(* IEC 61131-3 sources: Supremica/tests/ilprograms, 8 files *)

(* ---- arithmetictest.il ---- *)
(* Must test EQ before this.
 *)
PROGRAM ArithmeticTest
   VAR
	BB1, BB2, BB3 : BOOL;
	DD1, DD2, DD3 : DINT;
	RR1, RR2, RR3 : REAL;
	WW1, WW2, WW3 : WSTRING;
   END_VAR
   VAR
	Assert   : Asserter;
	(*Printing*)
	WPrintln : PrintlnWSTRING;
	DPrintln : PrintlnDINT;
	BPrintln : PrintlnBOOL;
	RPrintln : PrintlnREAL;
	WPrint   : PrintWSTRING;
	DPrint   : PrintDINT;
	BPrint   : PrintBOOL;
	RPrint   : PrintREAL;
   END_VAR

CAL WPrintln("Testing ADD")
	CAL Assert(TRUE,"här skall INGET fel ges")
	CAL Assert(FALSE,"här skall ett fel ges")
CAL WPrintln("Testing SUB")

CAL WPrintln("Testing MUL")

CAL WPrintln("Testing DIV")

CAL WPrintln("Testing MOD")

END_PROGRAM

FUNCTION_BLOCK Asserter
	VAR_IN_OUT
		result : BOOL;
		msg    : WSTRING;
	END_VAR
	VAR
		WPrintln : PrintlnWSTRING;
		WPrint   : PrintWSTRING;
	END_VAR
	LD result
	JMPC noerror
		CAL WPrint(output := "fdsf")
		(*CAL WPrint("Error: assertion not true! : ")*)
		(*CAL WPrintln(msg)*)
noerror:
END_FUNCTION_BLOCK

(*JAVA_BLOCKS for printing (no newline)*)
(*=====================================*)

JAVA_BLOCK JPrintWSTRING
	VAR_IN_OUT
		output: WSTRING;
	END_VAR
END_JAVA_BLOCK
FUNCTION_BLOCK PrintWSTRING
	VAR_IN_OUT
		output: WSTRING;
	END_VAR
	VAR
		jblock: JPrintWSTRING;
	END_VAR
	LD output
	ST jblock.output
	CAL jblock
END_FUNCTION_BLOCK

JAVA_BLOCK JPrintDINT
	VAR_IN_OUT
		output: DINT;
	END_VAR
END_JAVA_BLOCK
FUNCTION_BLOCK PrintDINT
	VAR_IN_OUT
		output: DINT;
	END_VAR
	VAR
		jblock: JPrintDINT;
	END_VAR
	LD output
	ST jblock.output
	CAL jblock
END_FUNCTION_BLOCK
JAVA_BLOCK JPrintREAL
	VAR_IN_OUT
		output:REAL;
	END_VAR
END_JAVA_BLOCK
FUNCTION_BLOCK PrintREAL
	VAR_IN_OUT
		output:REAL;
	END_VAR
	VAR
		jblock:JPrintREAL;
	END_VAR
	LD output
	ST jblock.output
	CAL jblock
END_FUNCTION_BLOCK

JAVA_BLOCK JPrintBOOL
	VAR_IN_OUT
		output: BOOL;
	END_VAR
END_JAVA_BLOCK
FUNCTION_BLOCK PrintBOOL
	VAR_IN_OUT
		output: BOOL;
	END_VAR
	VAR
		jblock: JPrintBOOL;
	END_VAR
	LD output
	ST jblock.output
	CAL jblock
END_FUNCTION_BLOCK

(*JAVA_BLOCKS for printing (newline)*)
(*=====================================*)

JAVA_BLOCK JPrintlnWSTRING
	VAR_IN_OUT
		output: WSTRING;
	END_VAR
END_JAVA_BLOCK
FUNCTION_BLOCK PrintlnWSTRING
	VAR_IN_OUT
		output: WSTRING;
	END_VAR
	VAR
		jblock: JPrintlnWSTRING;
	END_VAR
	LD output
	ST jblock.output
	CAL jblock
END_FUNCTION_BLOCK

JAVA_BLOCK JPrintlnDINT
	VAR_IN_OUT
		output: DINT;
	END_VAR
END_JAVA_BLOCK
FUNCTION_BLOCK PrintlnDINT
	VAR_IN_OUT
		output: DINT;
	END_VAR
	VAR
		jblock: JPrintlnDINT;
	END_VAR
	LD output
	ST jblock.output
	CAL jblock
END_FUNCTION_BLOCK

JAVA_BLOCK JPrintlnREAL
	VAR_IN_OUT
		output:REAL;
	END_VAR
END_JAVA_BLOCK
FUNCTION_BLOCK PrintlnREAL
	VAR_IN_OUT
		output:REAL;
	END_VAR
	VAR
		jblock:JPrintlnREAL;
	END_VAR
	LD output
	ST jblock.output
	CAL jblock
END_FUNCTION_BLOCK

JAVA_BLOCK JPrintlnBOOL
	VAR_IN_OUT
		output: BOOL;
	END_VAR
END_JAVA_BLOCK
FUNCTION_BLOCK PrintlnBOOL
	VAR_IN_OUT
		output: BOOL;
	END_VAR
	VAR
		jblock: JPrintlnBOOL;
	END_VAR
	LD output
	ST jblock.output
	CAL jblock
END_FUNCTION_BLOCK

(* ---- caltest.il ---- *)
(*JAVA_BLOCKS for printing (no newline)*)
(*=====================================*)

JAVA_BLOCK JPrintWSTRING
	VAR_IN_OUT
		output: WSTRING;
	END_VAR
END_JAVA_BLOCK
FUNCTION_BLOCK PrintWSTRING
	VAR_IN_OUT
		output: WSTRING;
	END_VAR
	VAR
		jblock: JPrintWSTRING;
	END_VAR
	LD output
	ST jblock.output
	CAL jblock
END_FUNCTION_BLOCK

JAVA_BLOCK JPrintDINT
	VAR_IN_OUT
		output: DINT;
	END_VAR
END_JAVA_BLOCK
FUNCTION_BLOCK PrintDINT
	VAR_IN_OUT
		output: DINT;
	END_VAR
	VAR
		jblock: JPrintDINT;
	END_VAR
	LD output
	ST jblock.output
	CAL jblock
END_FUNCTION_BLOCK

JAVA_BLOCK JPrintREAL
	VAR_IN_OUT
		output:REAL;
	END_VAR
END_JAVA_BLOCK
FUNCTION_BLOCK PrintREAL
	VAR_IN_OUT
		output:REAL;
	END_VAR
	VAR
		jblock:JPrintREAL;
	END_VAR
	LD output
	ST jblock.output
	CAL jblock
END_FUNCTION_BLOCK

JAVA_BLOCK JPrintBOOL
	VAR_IN_OUT
		output: BOOL;
	END_VAR
END_JAVA_BLOCK
FUNCTION_BLOCK PrintBOOL
	VAR_IN_OUT
		output: BOOL;
	END_VAR
	VAR
		jblock: JPrintBOOL;
	END_VAR
	LD output
	ST jblock.output
	CAL jblock
END_FUNCTION_BLOCK

(*JAVA_BLOCKS for printing (newline)*)
(*=====================================*)

JAVA_BLOCK JPrintlnWSTRING
	VAR_IN_OUT
		output: WSTRING;
	END_VAR
END_JAVA_BLOCK
FUNCTION_BLOCK PrintlnWSTRING
	VAR_IN_OUT
		output: WSTRING;
	END_VAR
	VAR
		jblock: JPrintlnWSTRING;
	END_VAR
	LD output
	ST jblock.output
	CAL jblock
END_FUNCTION_BLOCK

JAVA_BLOCK JPrintlnDINT
	VAR_IN_OUT
		output: DINT;
	END_VAR
END_JAVA_BLOCK
FUNCTION_BLOCK PrintlnDINT
	VAR_IN_OUT
		output: DINT;
	END_VAR
	VAR
		jblock: JPrintlnDINT;
	END_VAR
	LD output
	ST jblock.output
	CAL jblock
END_FUNCTION_BLOCK

JAVA_BLOCK JPrintlnREAL
	VAR_IN_OUT
		output:REAL;
	END_VAR
END_JAVA_BLOCK
FUNCTION_BLOCK PrintlnREAL
	VAR_IN_OUT
		output:REAL;
	END_VAR
	VAR
		jblock:JPrintlnREAL;
	END_VAR
	LD output
	ST jblock.output
	CAL jblock
END_FUNCTION_BLOCK

JAVA_BLOCK JPrintlnBOOL
	VAR_IN_OUT
		output: BOOL;
	END_VAR
END_JAVA_BLOCK
FUNCTION_BLOCK PrintlnBOOL
	VAR_IN_OUT
		output: BOOL;
	END_VAR
	VAR
		jblock: JPrintlnBOOL;
	END_VAR
	LD output
	ST jblock.output
	CAL jblock
END_FUNCTION_BLOCK

FUNCTION_BLOCK PrintlnWSTRING_DINT
	VAR_IN_OUT
		string: WSTRING;
		dint  : DINT;
	END_VAR
	VAR
		jblockWS: JPrintWSTRING;
		jblockD : JPrintlnDINT;
	END_VAR

	LD string
	ST jblockWS.output
	CAL jblockWS

	LD dint
	ST jblockD.output
	CAL jblockD
END_FUNCTION_BLOCK

FUNCTION_BLOCK DOUBLER
	VAR_IN_OUT
		A : DINT;
	END_VAR

	LD A
	ADD A

	ST A

END_FUNCTION_BLOCK

FUNCTION_BLOCK ADDER
	VAR_IN_OUT
		in_1 : DINT;
	    in_2 : DINT;
		out  : DINT;
	END_VAR

	LD in_1
	ADD in_2

	ST out

END_FUNCTION_BLOCK

FUNCTION_BLOCK ANDER
	VAR_IN_OUT
		in_1 : BOOL;
	    in_2 : BOOL;
		out  : BOOL;

	END_VAR

	LD in_1
	AND in_2
	ST out

END_FUNCTION_BLOCK

PROGRAM CALTEST
	VAR
		print_WS   : PrintWSTRING;
		print_DINT : PrintDINT;
		print_REAL : PrintREAL;
		print_BOOL : PrintBOOL;

		println_WS   : PrintlnWSTRING;
		println_DINT : PrintlnDINT;
		println_REAL : PrintlnREAL;
		println_BOOL : PrintlnBOOL;

		printlnWS_D  : PrintlnWSTRING_DINT;

      	doubler      : DOUBLER;
		adder        : ADDER;
		ander        : ANDER;

		N1           : DINT;
		N2           : DINT;
      	Result_DINT  : DINT;
		Result_BOOL  : BOOL;
	END_VAR
	VAR
		b AT %QX1 : BOOL;
	END_VAR

	LD FALSE
	ST %QX1

	LD %QX1
	ST Result_BOOL

	CAL println_BOOL(Result_BOOL)

	CAL println_BOOL(%QX1)

	LD DINT#10
	ST N1

	CAL printlnWS_D("Doubler input: ", N1)
    CAL doubler(N1)
	CAL printlnWS_D("Doubler output: ", doubler.A)

	CAL printlnWS_D("Doubler input: ", N1)
    CAL doubler(A:=N1)
	CAL printlnWS_D("Doubler output: ", doubler.A)

	CAL printlnWS_D("Doubler input: ", DINT#33)
    CAL doubler(DINT#33)
	CAL printlnWS_D("Doubler output: ", doubler.A)

	CAL printlnWS_D("Doubler input: ", DINT#33)
    CAL doubler(A:=DINT#33)
	CAL printlnWS_D("Doubler output: ", doubler.A)

	CAL adder(in_1:=DINT#100, in_2:=DINT#200, out=>Result_DINT)
	CAL println_DINT(Result_DINT)

	CAL ander(in_1:=FALSE, in_2:=TRUE, out=>%QX1)
	CAL println_BOOL(%QX1)

END_PROGRAM

(* ---- cmp_tests.il ---- *)
(*
Test av EQ, GT, GE, LT, LE, NE
*)

JAVA_BLOCK JPrintWSTRING
	VAR_IN_OUT
		output: WSTRING;
	END_VAR
END_JAVA_BLOCK
FUNCTION_BLOCK PrintWSTRING
	VAR_IN_OUT
		output: WSTRING;
	END_VAR
	VAR
		jblock: JPrintWSTRING;
	END_VAR
	LD output
	ST jblock.output
	CAL jblock
END_FUNCTION_BLOCK

JAVA_BLOCK JPrintDINT
	VAR_IN_OUT
		output: DINT;
	END_VAR
END_JAVA_BLOCK
FUNCTION_BLOCK PrintDINT
	VAR_IN_OUT
		output: DINT;
	END_VAR
	VAR
		jblock: JPrintDINT;
	END_VAR
	LD output
	ST jblock.output
	CAL jblock
END_FUNCTION_BLOCK
JAVA_BLOCK JPrintREAL
	VAR_IN_OUT
		output:REAL;
	END_VAR
END_JAVA_BLOCK
FUNCTION_BLOCK PrintREAL
	VAR_IN_OUT
		output:REAL;
	END_VAR
	VAR
		jblock:JPrintREAL;
	END_VAR
	LD output
	ST jblock.output
	CAL jblock
END_FUNCTION_BLOCK

JAVA_BLOCK JPrintBOOL
	VAR_IN_OUT
		output: BOOL;
	END_VAR
END_JAVA_BLOCK
FUNCTION_BLOCK PrintBOOL
	VAR_IN_OUT
		output: BOOL;
	END_VAR
	VAR
		jblock: JPrintBOOL;
	END_VAR
	LD output
	ST jblock.output
	CAL jblock
END_FUNCTION_BLOCK

JAVA_BLOCK JPrintlnWSTRING
	VAR_IN_OUT
		output: WSTRING;
	END_VAR
END_JAVA_BLOCK
FUNCTION_BLOCK PrintlnWSTRING
	VAR_IN_OUT
		output: WSTRING;
	END_VAR
	VAR
		jblock: JPrintlnWSTRING;
	END_VAR
	LD output
	ST jblock.output
	CAL jblock
END_FUNCTION_BLOCK

JAVA_BLOCK JPrintlnBOOL
	VAR_IN_OUT
		output: BOOL;
	END_VAR
END_JAVA_BLOCK
FUNCTION_BLOCK PrintlnBOOL
	VAR_IN_OUT
		output: BOOL;
	END_VAR
	VAR
		jblock: JPrintlnBOOL;
	END_VAR
	LD output
	ST jblock.output
	CAL jblock
END_FUNCTION_BLOCK

JAVA_BLOCK JPrintlnDINT
	VAR_IN_OUT
		output: DINT;
	END_VAR
END_JAVA_BLOCK
FUNCTION_BLOCK PrintlnDINT
	VAR_IN_OUT
		output: DINT;
	END_VAR
	VAR
		jblock: JPrintlnDINT;
	END_VAR
	LD output
	ST jblock.output
	CAL jblock
END_FUNCTION_BLOCK

JAVA_BLOCK JPrintlnREAL
	VAR_IN_OUT
		output:REAL;
	END_VAR
END_JAVA_BLOCK
FUNCTION_BLOCK PrintlnREAL
	VAR_IN_OUT
		output:REAL;
	END_VAR
	VAR
		jblock:JPrintlnREAL;
	END_VAR
	LD output
	ST jblock.output
	CAL jblock
END_FUNCTION_BLOCK

PROGRAM CMPtests
   VAR
	BB1, BB2, BB3 : BOOL;
	DD1, DD2, DD3 : DINT;
	RR1, RR2, RR3 : REAL;
	WW1, WW2, WW3 : WSTRING;
	PRINT_S : JPrintWSTRING;
	PRINT_B : JPrintBOOL;
	PRINT_I : JPrintDINT;
	PRINT_R : JPrintREAL;
	PRINTLN_S : JPrintlnWSTRING;
	PRINTLN_B : JPrintlnBOOL;
	PRINTLN_I : JPrintlnDINT;
	PRINTLN_R : JPrintlnREAL;
   END_VAR

	(*BOOL- jämför stack med variabel*)
	CAL PRINTLN_S(output:="EQ - BOOL")
(*T-T*)
	LD TRUE
	ST BB1
	LD TRUE
	EQ BB1
	ST BB2
	CAL PRINT_S(output:="?? true == ")
	CAL PRINTLN_B(output:=BB2)
(*T-F*)
	LD FALSE
	ST BB1
	LD TRUE
	EQ BB1
	ST BB2
	CAL PRINT_S(output:="?? false == ")
	CAL PRINTLN_B(output:=BB2)
(*F-T*)
	LD TRUE
	ST BB1
	LD FALSE
	EQ BB1
	ST BB2
	CAL PRINT_S(output:="?? false == ")
	CAL PRINTLN_B(output:=BB2)
(*F-F*)
	LD FALSE
	ST BB1
	LD FALSE
	EQ BB1
	ST BB2
	CAL PRINT_S(output:="?? true == ")
	CAL PRINTLN_B(output:=BB2)

	(*BOOL- jämför stack med konstant*)
(*T-T*)
	LD TRUE
	EQ TRUE
	ST BB2
	CAL PRINT_S(output:="?? true == ")
	CAL PRINTLN_B(output:=BB2)
(*T-F*)
	LD FALSE
	EQ TRUE
	ST BB2
	CAL PRINT_S(output:="?? false == ")
	CAL PRINTLN_B(output:=BB2)
(*F-T*)
	LD TRUE
	EQ FALSE
	ST BB2
	CAL PRINT_S(output:="?? false == ")
	CAL PRINTLN_B(output:=BB2)
(*F-F*)
	LD FALSE
	ST BB1
	LD FALSE
	EQ BB1
	ST BB2
	CAL PRINT_S(output:="?? true == ")
	CAL PRINTLN_B(output:=BB2)

	(*DINT - jämför stack med variabel*)
	CAL PRINTLN_S(output:="EQ - DINT")
(*1-1*)
	LD DINT#1
	ST DD1
	LD DINT#1
	EQ DD1
	ST BB2
	CAL PRINT_S(output:="?? true == ")
	CAL PRINTLN_B(output:=BB2)
(*2147483647 - 2147483647*)
	LD DINT#2147483647
	ST DD1
	LD DINT#2147483647
	EQ DD1
	ST BB2
	CAL PRINT_S(output:="?? true == ")
	CAL PRINTLN_B(output:=BB2)
(*-2147483647 - -2147483647*)
	LD DINT#-2147483647
	ST DD1
	LD DINT#-2147483647
	EQ DD1
	ST BB2
	CAL PRINT_S(output:="?? true == ")
	CAL PRINTLN_B(output:=BB2)
(*0 - 2147483647*)
	LD DINT#2147483647
	ST DD1
	LD DINT#0
	EQ DD1
	ST BB2
	CAL PRINT_S(output:="?? false == ")
	CAL PRINTLN_B(output:=BB2)
(*0 - -2147483647*)
	LD DINT#-2147483647
	ST DD1
	LD DINT#0
	EQ DD1
	ST BB2
	CAL PRINT_S(output:="?? false == ")
	CAL PRINTLN_B(output:=BB2)
(*-2147483647 - 0*)
	LD DINT#0
	ST DD1
	LD DINT#-2147483647
	EQ DD1
	ST BB2
	CAL PRINT_S(output:="?? false == ")
	CAL PRINTLN_B(output:=BB2)
(*2147483647 - 0*)
	LD DINT#0
	ST DD1
	LD DINT#2147483647
	EQ DD1
	ST BB2
	CAL PRINT_S(output:="?? false == ")
	CAL PRINTLN_B(output:=BB2)

	(*DINT- jämför stack med konstant*)
(*1-1*)
	LD DINT#1
	EQ DINT#1
	ST BB2
	CAL PRINT_S(output:="?? true == ")
	CAL PRINTLN_B(output:=BB2)
(*2147483647 - 2147483647*)
	LD DINT#2147483647
	EQ DINT#2147483647
	ST BB2
	CAL PRINT_S(output:="?? true == ")
	CAL PRINTLN_B(output:=BB2)
(*-2147483647 - -2147483647*)
	LD DINT#-2147483647
	EQ DINT#-2147483647
	ST BB2
	CAL PRINT_S(output:="?? true == ")
	CAL PRINTLN_B(output:=BB2)
(*0 - -2147483647*)
	LD DINT#2147483647
	EQ DINT#0
	ST BB2
	CAL PRINT_S(output:="?? false == ")
	CAL PRINTLN_B(output:=BB2)
(*0 - -2147483647*)
	LD DINT#-2147483647
	EQ DINT#0
	ST BB2
	CAL PRINT_S(output:="?? false == ")
	CAL PRINTLN_B(output:=BB2)
(*-2147483647 - 0*)
	LD DINT#0
	EQ DINT#-2147483647
	ST BB2
	CAL PRINT_S(output:="?? false == ")
	CAL PRINTLN_B(output:=BB2)
(*2147483647 - 0*)
	LD DINT#0
	EQ DINT#2147483647
	ST BB2
	CAL PRINT_S(output:="?? false == ")
	CAL PRINTLN_B(output:=BB2)

	(*EQ - REAL - jämför stack med variabel*)
	CAL PRINTLN_S(output:="EQ - REAL")
(*1.0 - 1.0*)
	LD REAL#1.0
	ST RR1
	LD REAL#1.0
	EQ RR1
	ST BB2
	CAL PRINT_S(output:="?? true == ")
	CAL PRINTLN_B(output:=BB2)
(*3.4028235E38 - 3.4028235E38*)
	LD REAL#3.4028235E38
	ST RR1
	LD REAL#3.4028235E38
	EQ RR1
	ST BB2
	CAL PRINT_S(output:="?? true == ")
	CAL PRINTLN_B(output:=BB2)
(*1.4E-45 - 1.4E-45*)
	LD REAL#1.4E-45
	ST RR1
	LD REAL#1.4E-45
	EQ RR1
	ST BB2
	CAL PRINT_S(output:="?? true == ")
	CAL PRINTLN_B(output:=BB2)
(*0 - 3.4028235E38*)
	LD REAL#3.4028235E38
	ST RR1
	LD REAL#0.0
	EQ RR1
	ST BB2
	CAL PRINT_S(output:="?? false == ")
	CAL PRINTLN_B(output:=BB2)
(*0 - 1.4E-45*)
	LD REAL#1.4E-45
	ST RR1
	LD REAL#0.0
	EQ RR1
	ST BB2
	CAL PRINT_S(output:="?? false == ")
	CAL PRINTLN_B(output:=BB2)
(*1.4E-45 - 0*)
	LD REAL#0.0
	ST RR1
	LD REAL#1.4E-45
	EQ RR1
	ST BB2
	CAL PRINT_S(output:="?? false == ")
	CAL PRINTLN_B(output:=BB2)
(*3.4028235E38 - 0*)
	LD REAL#0.0
	ST RR1
	LD REAL#3.4028235E38
	EQ RR1
	ST BB2
	CAL PRINT_S(output:="?? false == ")
	CAL PRINTLN_B(output:=BB2)

	(*EQ - REAL- jämför stack med konstant*)
(*1-1*)
	LD REAL#1.0
	EQ REAL#1.0
	ST BB2
	CAL PRINT_S(output:="?? true == ")
	CAL PRINTLN_B(output:=BB2)
(*3.4028235E38 - 3.4028235E38*)
	LD REAL#3.4028235E38
	EQ REAL#3.4028235E38
	ST BB2
	CAL PRINT_S(output:="?? true == ")
	CAL PRINTLN_B(output:=BB2)
(*1.4E-45 - 1.4E-45*)
	LD REAL#1.4E-45
	EQ REAL#1.4E-45
	ST BB2
	CAL PRINT_S(output:="?? true == ")
	CAL PRINTLN_B(output:=BB2)
(*0 - 3.4028235E38*)
	LD REAL#3.4028235E38
	EQ REAL#0.0
	ST BB2
	CAL PRINT_S(output:="?? false == ")
	CAL PRINTLN_B(output:=BB2)
(*0 - 1.4E-45*)
	LD REAL#1.4E-45
	EQ REAL#0.0
	ST BB2
	CAL PRINT_S(output:="?? false == ")
	CAL PRINTLN_B(output:=BB2)
(*1.4E-45 - 0*)
	LD REAL#0.0
	EQ REAL#1.4E-45
	ST BB2
	CAL PRINT_S(output:="?? false == ")
	CAL PRINTLN_B(output:=BB2)
(*3.4028235E38 - 0*)
	LD REAL#0.0
	EQ REAL#3.4028235E38
	ST BB2
	CAL PRINT_S(output:="?? false == ")
	CAL PRINTLN_B(output:=BB2)

(******************************************************************)

	(*GT - DINT - jämför stack med variabel*)
	CAL PRINTLN_S(output:="GT - DINT")
(*1-1*)
	LD DINT#1
	ST DD1
	LD DINT#1
	GT DD1
	ST BB2
	CAL PRINT_S(output:="?? false == ")
	CAL PRINTLN_B(output:=BB2)
(*2147483647 - 2147483647*)
	LD DINT#2147483647
	ST DD1
	LD DINT#2147483647
	GT DD1
	ST BB2
	CAL PRINT_S(output:="?? false == ")
	CAL PRINTLN_B(output:=BB2)
(*-2147483647 - -2147483647*)
	LD DINT#-2147483647
	ST DD1
	LD DINT#-2147483647
	GT DD1
	ST BB2
	CAL PRINT_S(output:="?? false == ")
	CAL PRINTLN_B(output:=BB2)
(*0 - 2147483647*)
	LD DINT#2147483647
	ST DD1
	LD DINT#0
	GT DD1
	ST BB2
	CAL PRINT_S(output:="?? false == ")
	CAL PRINTLN_B(output:=BB2)
(*0 - -2147483647*)
	LD DINT#-2147483647
	ST DD1
	LD DINT#0
	GT DD1
	ST BB2
	CAL PRINT_S(output:="?? true == ")
	CAL PRINTLN_B(output:=BB2)
(*-2147483647 - 0*)
	LD DINT#0
	ST DD1
	LD DINT#-2147483647
	GT DD1
	ST BB2
	CAL PRINT_S(output:="?? false == ")
	CAL PRINTLN_B(output:=BB2)
(*2147483647 - 0*)
	LD DINT#0
	ST DD1
	LD DINT#2147483647
	GT DD1
	ST BB2
	CAL PRINT_S(output:="?? true == ")
	CAL PRINTLN_B(output:=BB2)

	(*GT - DINT - jämför stack med konstant*)
(*1-1*)
	LD DINT#1
	GT DINT#1
	ST BB2
	CAL PRINT_S(output:="?? false == ")
	CAL PRINTLN_B(output:=BB2)
(*2147483647 - 2147483647*)
	LD DINT#2147483647
	GT DINT#2147483647
	ST BB2
	CAL PRINT_S(output:="?? false == ")
	CAL PRINTLN_B(output:=BB2)
(*-2147483647 - -2147483647*)
	LD DINT#-2147483647
	GT DINT#-2147483647
	ST BB2
	CAL PRINT_S(output:="?? false == ")
	CAL PRINTLN_B(output:=BB2)
(*2147483647 - 0*)
	LD DINT#2147483647
	GT DINT#0
	ST BB2
	CAL PRINT_S(output:="?? true == ")
	CAL PRINTLN_B(output:=BB2)
(*-2147483647 - 0*)
	LD DINT#-2147483647
	GT DINT#0
	ST BB2
	CAL PRINT_S(output:="?? false == ")
	CAL PRINTLN_B(output:=BB2)
(*0 - -2147483647*)
	LD DINT#0
	GT DINT#-2147483647
	ST BB2
	CAL PRINT_S(output:="?? true == ")
	CAL PRINTLN_B(output:=BB2)
(*0 - 2147483647*)
	LD DINT#0
	GT DINT#2147483647
	ST BB2
	CAL PRINT_S(output:="?? false == ")
	CAL PRINTLN_B(output:=BB2)

	(*GT - REAL - jämför stack med variabel*)
	CAL PRINTLN_S(output:="GT - REAL")
(*1.0 - 1.0*)
	LD REAL#1.0
	ST RR1
	LD REAL#1.0
	GT RR1
	ST BB2
	CAL PRINT_S(output:="?? false == ")
	CAL PRINTLN_B(output:=BB2)
(*3.4028235E38 - 3.4028235E38*)
	LD REAL#3.4028235E38
	ST RR1
	LD REAL#3.4028235E38
	GT RR1
	ST BB2
	CAL PRINT_S(output:="?? false == ")
	CAL PRINTLN_B(output:=BB2)
(*1.4E-45 - 1.4E-45*)
	LD REAL#1.4E-45
	ST RR1
	LD REAL#1.4E-45
	GT RR1
	ST BB2
	CAL PRINT_S(output:="?? false == ")
	CAL PRINTLN_B(output:=BB2)
(*0 - 3.4028235E38*)
	LD REAL#3.4028235E38
	ST RR1
	LD REAL#0.0
	GT RR1
	ST BB2
	CAL PRINT_S(output:="?? false == ")
	CAL PRINTLN_B(output:=BB2)
(*0 - 1.4E-45*)
	LD REAL#1.4E-45
	ST RR1
	LD REAL#0.0
	GT RR1
	ST BB2
	CAL PRINT_S(output:="?? false == ")
	CAL PRINTLN_B(output:=BB2)
(*1.4E-45 - 0*)
	LD REAL#0.0
	ST RR1
	LD REAL#1.4E-45
	GT RR1
	ST BB2
	CAL PRINT_S(output:="?? true == ")
	CAL PRINTLN_B(output:=BB2)
(*3.4028235E38 - 0*)
	LD REAL#0.0
	ST RR1
	LD REAL#3.4028235E38
	GT RR1
	ST BB2
	CAL PRINT_S(output:="?? true == ")
	CAL PRINTLN_B(output:=BB2)

	(*GT - REAL - jämför stack med konstant*)
(*1-1*)
	LD REAL#1.0
	GT REAL#1.0
	ST BB2
	CAL PRINT_S(output:="?? false == ")
	CAL PRINTLN_B(output:=BB2)
(*3.4028235E38 - 3.4028235E38*)
	LD REAL#3.4028235E38
	GT REAL#3.4028235E38
	ST BB2
	CAL PRINT_S(output:="?? false == ")
	CAL PRINTLN_B(output:=BB2)
(*1.4E-45 - 1.4E-45*)
	LD REAL#1.4E-45
	GT REAL#1.4E-45
	ST BB2
	CAL PRINT_S(output:="?? false == ")
	CAL PRINTLN_B(output:=BB2)
(*3.4028235E38 - 0*)
	LD REAL#3.4028235E38
	GT REAL#0.0
	ST BB2
	CAL PRINT_S(output:="?? true == ")
	CAL PRINTLN_B(output:=BB2)
(*1.4E-45 - 0*)
	LD REAL#1.4E-45
	GT REAL#0.0
	ST BB2
	CAL PRINT_S(output:="?? true == ")
	CAL PRINTLN_B(output:=BB2)
(*0 - 1.4E-45*)
	LD REAL#0.0
	GT REAL#1.4E-45
	ST BB2
	CAL PRINT_S(output:="?? false == ")
	CAL PRINTLN_B(output:=BB2)
(*0 - 3.4028235E38*)
	LD REAL#0.0
	GT REAL#3.4028235E38
	ST BB2
	CAL PRINT_S(output:="?? false == ")
	CAL PRINTLN_B(output:=BB2)

(*****************************************************************)

	(*GE - DINT - jämför stack med variabel*)
	CAL PRINTLN_S(output:="GE - DINT")
(*1-1*)
	LD DINT#1
	ST DD1
	LD DINT#1
	GE DD1
	ST BB2
	CAL PRINT_S(output:="?? true == ")
	CAL PRINTLN_B(output:=BB2)
(*2147483647 - 2147483647*)
	LD DINT#2147483647
	ST DD1
	LD DINT#2147483647
	GE DD1
	ST BB2
	CAL PRINT_S(output:="?? true == ")
	CAL PRINTLN_B(output:=BB2)
(*-2147483647 - -2147483647*)
	LD DINT#-2147483647
	ST DD1
	LD DINT#-2147483647
	GE DD1
	ST BB2
	CAL PRINT_S(output:="?? true == ")
	CAL PRINTLN_B(output:=BB2)
(*0 - 2147483647*)
	LD DINT#2147483647
	ST DD1
	LD DINT#0
	GE DD1
	ST BB2
	CAL PRINT_S(output:="?? false == ")
	CAL PRINTLN_B(output:=BB2)
(*0 - -2147483647*)
	LD DINT#-2147483647
	ST DD1
	LD DINT#0
	GE DD1
	ST BB2
	CAL PRINT_S(output:="?? true == ")
	CAL PRINTLN_B(output:=BB2)
(*-2147483647 - 0*)
	LD DINT#0
	ST DD1
	LD DINT#-2147483647
	GE DD1
	ST BB2
	CAL PRINT_S(output:="?? false == ")
	CAL PRINTLN_B(output:=BB2)
(*2147483647 - 0*)
	LD DINT#0
	ST DD1
	LD DINT#2147483647
	GE DD1
	ST BB2
	CAL PRINT_S(output:="?? true == ")
	CAL PRINTLN_B(output:=BB2)

	(*GE - DINT - jämför stack med konstant*)
(*1-1*)
	LD DINT#1
	GE DINT#1
	ST BB2
	CAL PRINT_S(output:="?? true == ")
	CAL PRINTLN_B(output:=BB2)
(*2147483647 - 2147483647*)
	LD DINT#2147483647
	GE DINT#2147483647
	ST BB2
	CAL PRINT_S(output:="?? true == ")
	CAL PRINTLN_B(output:=BB2)
(*-2147483647 - -2147483647*)
	LD DINT#-2147483647
	GE DINT#-2147483647
	ST BB2
	CAL PRINT_S(output:="?? true == ")
	CAL PRINTLN_B(output:=BB2)
(*2147483647 - 0*)
	LD DINT#2147483647
	GE DINT#0
	ST BB2
	CAL PRINT_S(output:="?? true == ")
	CAL PRINTLN_B(output:=BB2)
(*-2147483647 - 0*)
	LD DINT#-2147483647
	GE DINT#0
	ST BB2
	CAL PRINT_S(output:="?? false == ")
	CAL PRINTLN_B(output:=BB2)
(*0 - -2147483647*)
	LD DINT#0
	GE DINT#-2147483647
	ST BB2
	CAL PRINT_S(output:="?? true == ")
	CAL PRINTLN_B(output:=BB2)
(*0 - 2147483647*)
	LD DINT#0
	GE DINT#2147483647
	ST BB2
	CAL PRINT_S(output:="?? false == ")
	CAL PRINTLN_B(output:=BB2)

	(*GE - REAL - jämför stack med variabel*)
	CAL PRINTLN_S(output:="GE - REAL")
(*1.0 - 1.0*)
	LD REAL#1.0
	ST RR1
	LD REAL#1.0
	GE RR1
	ST BB2
	CAL PRINT_S(output:="?? true == ")
	CAL PRINTLN_B(output:=BB2)
(*3.4028235E38 - 3.4028235E38*)
	LD REAL#3.4028235E38
	ST RR1
	LD REAL#3.4028235E38
	GE RR1
	ST BB2
	CAL PRINT_S(output:="?? true == ")
	CAL PRINTLN_B(output:=BB2)
(*1.4E-45 - 1.4E-45*)
	LD REAL#1.4E-45
	ST RR1
	LD REAL#1.4E-45
	GE RR1
	ST BB2
	CAL PRINT_S(output:="?? true == ")
	CAL PRINTLN_B(output:=BB2)
(*0 - 3.4028235E38*)
	LD REAL#3.4028235E38
	ST RR1
	LD REAL#0.0
	GE RR1
	ST BB2
	CAL PRINT_S(output:="?? false == ")
	CAL PRINTLN_B(output:=BB2)
(*0 - 1.4E-45*)
	LD REAL#1.4E-45
	ST RR1
	LD REAL#0.0
	GE RR1
	ST BB2
	CAL PRINT_S(output:="?? false == ")
	CAL PRINTLN_B(output:=BB2)
(*1.4E-45 - 0*)
	LD REAL#0.0
	ST RR1
	LD REAL#1.4E-45
	GE RR1
	ST BB2
	CAL PRINT_S(output:="?? true == ")
	CAL PRINTLN_B(output:=BB2)
(*3.4028235E38 - 0*)
	LD REAL#0.0
	ST RR1
	LD REAL#3.4028235E38
	GE RR1
	ST BB2
	CAL PRINT_S(output:="?? true == ")
	CAL PRINTLN_B(output:=BB2)

	(*GE - REAL - jämför stack med konstant*)
(*1-1*)
	LD REAL#1.0
	GE REAL#1.0
	ST BB2
	CAL PRINT_S(output:="?? true == ")
	CAL PRINTLN_B(output:=BB2)
(*3.4028235E38 - 3.4028235E38*)
	LD REAL#3.4028235E38
	GE REAL#3.4028235E38
	ST BB2
	CAL PRINT_S(output:="?? true == ")
	CAL PRINTLN_B(output:=BB2)
(*1.4E-45 - 1.4E-45*)
	LD REAL#1.4E-45
	GE REAL#1.4E-45
	ST BB2
	CAL PRINT_S(output:="?? true == ")
	CAL PRINTLN_B(output:=BB2)
(*3.4028235E38 - 0*)
	LD REAL#3.4028235E38
	GE REAL#0.0
	ST BB2
	CAL PRINT_S(output:="?? true == ")
	CAL PRINTLN_B(output:=BB2)
(*1.4E-45 - 0*)
	LD REAL#1.4E-45
	GE REAL#0.0
	ST BB2
	CAL PRINT_S(output:="?? true == ")
	CAL PRINTLN_B(output:=BB2)
(*0 - 1.4E-45*)
	LD REAL#0.0
	GE REAL#1.4E-45
	ST BB2
	CAL PRINT_S(output:="?? false == ")
	CAL PRINTLN_B(output:=BB2)
(*0 - 3.4028235E38*)
	LD REAL#0.0
	GE REAL#3.4028235E38
	ST BB2
	CAL PRINT_S(output:="?? false == ")
	CAL PRINTLN_B(output:=BB2)

(******************************************************************)

	(*LT - DINT - jämför stack med variabel*)
	CAL PRINTLN_S(output:="LT - DINT")
(*1-1*)
	LD DINT#1
	ST DD1
	LD DINT#1
	LT DD1
	ST BB2
	CAL PRINT_S(output:="?? false == ")
	CAL PRINTLN_B(output:=BB2)
(*2147483647 - 2147483647*)
	LD DINT#2147483647
	ST DD1
	LD DINT#2147483647
	LT DD1
	ST BB2
	CAL PRINT_S(output:="?? false == ")
	CAL PRINTLN_B(output:=BB2)
(*-2147483647 - -2147483647*)
	LD DINT#-2147483647
	ST DD1
	LD DINT#-2147483647
	LT DD1
	ST BB2
	CAL PRINT_S(output:="?? false == ")
	CAL PRINTLN_B(output:=BB2)
(*0 - 2147483647*)
	LD DINT#2147483647
	ST DD1
	LD DINT#0
	LT DD1
	ST BB2
	CAL PRINT_S(output:="?? true == ")
	CAL PRINTLN_B(output:=BB2)
(*0 - -2147483647*)
	LD DINT#-2147483647
	ST DD1
	LD DINT#0
	LT DD1
	ST BB2
	CAL PRINT_S(output:="?? false == ")
	CAL PRINTLN_B(output:=BB2)
(*-2147483647 - 0*)
	LD DINT#0
	ST DD1
	LD DINT#-2147483647
	LT DD1
	ST BB2
	CAL PRINT_S(output:="?? true == ")
	CAL PRINTLN_B(output:=BB2)
(*2147483647 - 0*)
	LD DINT#0
	ST DD1
	LD DINT#2147483647
	LT DD1
	ST BB2
	CAL PRINT_S(output:="?? false == ")
	CAL PRINTLN_B(output:=BB2)

	(*LT - DINT - jämför stack med konstant*)
(*1-1*)
	LD DINT#1
	LT DINT#1
	ST BB2
	CAL PRINT_S(output:="?? false == ")
	CAL PRINTLN_B(output:=BB2)
(*2147483647 - 2147483647*)
	LD DINT#2147483647
	LT DINT#2147483647
	ST BB2
	CAL PRINT_S(output:="?? false == ")
	CAL PRINTLN_B(output:=BB2)
(*-2147483647 - -2147483647*)
	LD DINT#-2147483647
	LT DINT#-2147483647
	ST BB2
	CAL PRINT_S(output:="?? false == ")
	CAL PRINTLN_B(output:=BB2)
(*2147483647 - 0*)
	LD DINT#2147483647
	LT DINT#0
	ST BB2
	CAL PRINT_S(output:="?? false == ")
	CAL PRINTLN_B(output:=BB2)
(*-2147483647 - 0*)
	LD DINT#-2147483647
	LT DINT#0
	ST BB2
	CAL PRINT_S(output:="?? true == ")
	CAL PRINTLN_B(output:=BB2)
(*0 - -2147483647*)
	LD DINT#0
	LT DINT#-2147483647
	ST BB2
	CAL PRINT_S(output:="?? false == ")
	CAL PRINTLN_B(output:=BB2)
(*0 - 2147483647*)
	LD DINT#0
	LT DINT#2147483647
	ST BB2
	CAL PRINT_S(output:="?? true == ")
	CAL PRINTLN_B(output:=BB2)

	(*LT - REAL - jämför stack med variabel*)
	CAL PRINTLN_S(output:="LT - REAL")
(*1.0 - 1.0*)
	LD REAL#1.0
	ST RR1
	LD REAL#1.0
	LT RR1
	ST BB2
	CAL PRINT_S(output:="?? false == ")
	CAL PRINTLN_B(output:=BB2)
(*3.4028235E38 - 3.4028235E38*)
	LD REAL#3.4028235E38
	ST RR1
	LD REAL#3.4028235E38
	LT RR1
	ST BB2
	CAL PRINT_S(output:="?? false == ")
	CAL PRINTLN_B(output:=BB2)
(*1.4E-45 - 1.4E-45*)
	LD REAL#1.4E-45
	ST RR1
	LD REAL#1.4E-45
	LT RR1
	ST BB2
	CAL PRINT_S(output:="?? false == ")
	CAL PRINTLN_B(output:=BB2)
(*0 - 3.4028235E38*)
	LD REAL#3.4028235E38
	ST RR1
	LD REAL#0.0
	LT RR1
	ST BB2
	CAL PRINT_S(output:="?? true == ")
	CAL PRINTLN_B(output:=BB2)
(*0 - 1.4E-45*)
	LD REAL#1.4E-45
	ST RR1
	LD REAL#0.0
	LT RR1
	ST BB2
	CAL PRINT_S(output:="?? true == ")
	CAL PRINTLN_B(output:=BB2)
(*1.4E-45 - 0*)
	LD REAL#0.0
	ST RR1
	LD REAL#1.4E-45
	LT RR1
	ST BB2
	CAL PRINT_S(output:="?? false == ")
	CAL PRINTLN_B(output:=BB2)
(*3.4028235E38 - 0*)
	LD REAL#0.0
	ST RR1
	LD REAL#3.4028235E38
	LT RR1
	ST BB2
	CAL PRINT_S(output:="?? false == ")
	CAL PRINTLN_B(output:=BB2)

	(*LT - REAL - jämför stack med konstant*)
(*1-1*)
	LD REAL#1.0
	LT REAL#1.0
	ST BB2
	CAL PRINT_S(output:="?? false == ")
	CAL PRINTLN_B(output:=BB2)
(*3.4028235E38 - 3.4028235E38*)
	LD REAL#3.4028235E38
	LT REAL#3.4028235E38
	ST BB2
	CAL PRINT_S(output:="?? false == ")
	CAL PRINTLN_B(output:=BB2)
(*1.4E-45 - 1.4E-45*)
	LD REAL#1.4E-45
	LT REAL#1.4E-45
	ST BB2
	CAL PRINT_S(output:="?? false == ")
	CAL PRINTLN_B(output:=BB2)
(*3.4028235E38 - 0*)
	LD REAL#3.4028235E38
	LT REAL#0.0
	ST BB2
	CAL PRINT_S(output:="?? false == ")
	CAL PRINTLN_B(output:=BB2)
(*1.4E-45 - 0*)
	LD REAL#1.4E-45
	LT REAL#0.0
	ST BB2
	CAL PRINT_S(output:="?? false == ")
	CAL PRINTLN_B(output:=BB2)
(*0 - 1.4E-45*)
	LD REAL#0.0
	LT REAL#1.4E-45
	ST BB2
	CAL PRINT_S(output:="?? true == ")
	CAL PRINTLN_B(output:=BB2)
(*0 - 3.4028235E38*)
	LD REAL#0.0
	LT REAL#3.4028235E38
	ST BB2
	CAL PRINT_S(output:="?? true == ")
	CAL PRINTLN_B(output:=BB2)

(******************************************************************)

	(*LE - DINT - jämför stack med variabel*)
	CAL PRINTLN_S(output:="LE - DINT")
(*1-1*)
	LD DINT#1
	ST DD1
	LD DINT#1
	LE DD1
	ST BB2
	CAL PRINT_S(output:="?? true == ")
	CAL PRINTLN_B(output:=BB2)
(*2147483647 - 2147483647*)
	LD DINT#2147483647
	ST DD1
	LD DINT#2147483647
	LE DD1
	ST BB2
	CAL PRINT_S(output:="?? true == ")
	CAL PRINTLN_B(output:=BB2)
(*-2147483647 - -2147483647*)
	LD DINT#-2147483647
	ST DD1
	LD DINT#-2147483647
	LE DD1
	ST BB2
	CAL PRINT_S(output:="?? true == ")
	CAL PRINTLN_B(output:=BB2)
(*0 - 2147483647*)
	LD DINT#2147483647
	ST DD1
	LD DINT#0
	LE DD1
	ST BB2
	CAL PRINT_S(output:="?? true == ")
	CAL PRINTLN_B(output:=BB2)
(*0 - -2147483647*)
	LD DINT#-2147483647
	ST DD1
	LD DINT#0
	LE DD1
	ST BB2
	CAL PRINT_S(output:="?? false == ")
	CAL PRINTLN_B(output:=BB2)
(*-2147483647 - 0*)
	LD DINT#0
	ST DD1
	LD DINT#-2147483647
	LE DD1
	ST BB2
	CAL PRINT_S(output:="?? true == ")
	CAL PRINTLN_B(output:=BB2)
(*2147483647 - 0*)
	LD DINT#0
	ST DD1
	LD DINT#2147483647
	LE DD1
	ST BB2
	CAL PRINT_S(output:="?? false == ")
	CAL PRINTLN_B(output:=BB2)

	(*LE - DINT - jämför stack med konstant*)
(*1-1*)
	LD DINT#1
	LE DINT#1
	ST BB2
	CAL PRINT_S(output:="?? true == ")
	CAL PRINTLN_B(output:=BB2)
(*2147483647 - 2147483647*)
	LD DINT#2147483647
	LE DINT#2147483647
	ST BB2
	CAL PRINT_S(output:="?? true == ")
	CAL PRINTLN_B(output:=BB2)
(*-2147483647 - -2147483647*)
	LD DINT#-2147483647
	LE DINT#-2147483647
	ST BB2
	CAL PRINT_S(output:="?? true == ")
	CAL PRINTLN_B(output:=BB2)
(*2147483647 - 0*)
	LD DINT#2147483647
	LE DINT#0
	ST BB2
	CAL PRINT_S(output:="?? false == ")
	CAL PRINTLN_B(output:=BB2)
(*-2147483647 - 0*)
	LD DINT#-2147483647
	LE DINT#0
	ST BB2
	CAL PRINT_S(output:="?? true == ")
	CAL PRINTLN_B(output:=BB2)
(*0 - -2147483647*)
	LD DINT#0
	LE DINT#-2147483647
	ST BB2
	CAL PRINT_S(output:="?? false == ")
	CAL PRINTLN_B(output:=BB2)
(*0 - 2147483647*)
	LD DINT#0
	LE DINT#2147483647
	ST BB2
	CAL PRINT_S(output:="?? true == ")
	CAL PRINTLN_B(output:=BB2)

	(*LE - REAL - jämför stack med variabel*)
	CAL PRINTLN_S(output:="LE - REAL")
(*1.0 - 1.0*)
	LD REAL#1.0
	ST RR1
	LD REAL#1.0
	LE RR1
	ST BB2
	CAL PRINT_S(output:="?? true == ")
	CAL PRINTLN_B(output:=BB2)
(*3.4028235E38 - 3.4028235E38*)
	LD REAL#3.4028235E38
	ST RR1
	LD REAL#3.4028235E38
	LE RR1
	ST BB2
	CAL PRINT_S(output:="?? true == ")
	CAL PRINTLN_B(output:=BB2)
(*1.4E-45 - 1.4E-45*)
	LD REAL#1.4E-45
	ST RR1
	LD REAL#1.4E-45
	LE RR1
	ST BB2
	CAL PRINT_S(output:="?? true == ")
	CAL PRINTLN_B(output:=BB2)
(*0 - 3.4028235E38*)
	LD REAL#3.4028235E38
	ST RR1
	LD REAL#0.0
	LE RR1
	ST BB2
	CAL PRINT_S(output:="?? true == ")
	CAL PRINTLN_B(output:=BB2)
(*0 - 1.4E-45*)
	LD REAL#1.4E-45
	ST RR1
	LD REAL#0.0
	LE RR1
	ST BB2
	CAL PRINT_S(output:="?? true == ")
	CAL PRINTLN_B(output:=BB2)
(*1.4E-45 - 0*)
	LD REAL#0.0
	ST RR1
	LD REAL#1.4E-45
	LE RR1
	ST BB2
	CAL PRINT_S(output:="?? false == ")
	CAL PRINTLN_B(output:=BB2)
(*3.4028235E38 - 0*)
	LD REAL#0.0
	ST RR1
	LD REAL#3.4028235E38
	LE RR1
	ST BB2
	CAL PRINT_S(output:="?? false == ")
	CAL PRINTLN_B(output:=BB2)

	(*LE - REAL - jämför stack med konstant*)
(*1-1*)
	LD REAL#1.0
	LE REAL#1.0
	ST BB2
	CAL PRINT_S(output:="?? true == ")
	CAL PRINTLN_B(output:=BB2)
(*3.4028235E38 - 3.4028235E38*)
	LD REAL#3.4028235E38
	LE REAL#3.4028235E38
	ST BB2
	CAL PRINT_S(output:="?? true == ")
	CAL PRINTLN_B(output:=BB2)
(*1.4E-45 - 1.4E-45*)
	LD REAL#1.4E-45
	LE REAL#1.4E-45
	ST BB2
	CAL PRINT_S(output:="?? true == ")
	CAL PRINTLN_B(output:=BB2)
(*3.4028235E38 - 0*)
	LD REAL#3.4028235E38
	LE REAL#0.0
	ST BB2
	CAL PRINT_S(output:="?? false == ")
	CAL PRINTLN_B(output:=BB2)
(*1.4E-45 - 0*)
	LD REAL#1.4E-45
	LE REAL#0.0
	ST BB2
	CAL PRINT_S(output:="?? false == ")
	CAL PRINTLN_B(output:=BB2)
(*0 - 1.4E-45*)
	LD REAL#0.0
	LE REAL#1.4E-45
	ST BB2
	CAL PRINT_S(output:="?? true == ")
	CAL PRINTLN_B(output:=BB2)
(*0 - 3.4028235E38*)
	LD REAL#0.0
	LE REAL#3.4028235E38
	ST BB2
	CAL PRINT_S(output:="?? true == ")
	CAL PRINTLN_B(output:=BB2)

(******************************************************************)

	CAL PRINTLN_S(output:="NE - BOOL")
(*T-T*)
	LD TRUE
	ST BB1
	LD TRUE
	NE BB1
	ST BB2
	CAL PRINT_S(output:="?? false == ")
	CAL PRINTLN_B(output:=BB2)
(*T-F*)
	LD FALSE
	ST BB1
	LD TRUE
	NE BB1
	ST BB2
	CAL PRINT_S(output:="?? true == ")
	CAL PRINTLN_B(output:=BB2)
(*F-T*)
	LD TRUE
	ST BB1
	LD FALSE
	NE BB1
	ST BB2
	CAL PRINT_S(output:="?? true == ")
	CAL PRINTLN_B(output:=BB2)
(*F-F*)
	LD FALSE
	ST BB1
	LD FALSE
	NE BB1
	ST BB2
	CAL PRINT_S(output:="?? false == ")
	CAL PRINTLN_B(output:=BB2)

	(*BOOL- jämför stack med konstant*)
(*T-T*)
	LD TRUE
	NE TRUE
	ST BB2
	CAL PRINT_S(output:="?? false == ")
	CAL PRINTLN_B(output:=BB2)
(*T-F*)
	LD FALSE
	NE TRUE
	ST BB2
	CAL PRINT_S(output:="?? true == ")
	CAL PRINTLN_B(output:=BB2)
(*F-T*)
	LD TRUE
	NE FALSE
	ST BB2
	CAL PRINT_S(output:="?? true == ")
	CAL PRINTLN_B(output:=BB2)
(*F-F*)
	LD FALSE
	ST BB1
	LD FALSE
	NE BB1
	ST BB2
	CAL PRINT_S(output:="?? false == ")
	CAL PRINTLN_B(output:=BB2)

	(*NE - DINT - jämför stack med variabel*)
	CAL PRINTLN_S(output:="NE - DINT")
(*1-1*)
	LD DINT#1
	ST DD1
	LD DINT#1
	NE DD1
	ST BB2
	CAL PRINT_S(output:="?? false == ")
	CAL PRINTLN_B(output:=BB2)
(*2147483647 - 2147483647*)
	LD DINT#2147483647
	ST DD1
	LD DINT#2147483647
	NE DD1
	ST BB2
	CAL PRINT_S(output:="?? false == ")
	CAL PRINTLN_B(output:=BB2)
(*-2147483647 - -2147483647*)
	LD DINT#-2147483647
	ST DD1
	LD DINT#-2147483647
	NE DD1
	ST BB2
	CAL PRINT_S(output:="?? false == ")
	CAL PRINTLN_B(output:=BB2)
(*0 - 2147483647*)
	LD DINT#2147483647
	ST DD1
	LD DINT#0
	NE DD1
	ST BB2
	CAL PRINT_S(output:="?? true == ")
	CAL PRINTLN_B(output:=BB2)
(*0 - -2147483647*)
	LD DINT#-2147483647
	ST DD1
	LD DINT#0
	NE DD1
	ST BB2
	CAL PRINT_S(output:="?? true == ")
	CAL PRINTLN_B(output:=BB2)
(*-2147483647 - 0*)
	LD DINT#0
	ST DD1
	LD DINT#-2147483647
	NE DD1
	ST BB2
	CAL PRINT_S(output:="?? true == ")
	CAL PRINTLN_B(output:=BB2)
(*2147483647 - 0*)
	LD DINT#0
	ST DD1
	LD DINT#2147483647
	NE DD1
	ST BB2
	CAL PRINT_S(output:="?? true == ")
	CAL PRINTLN_B(output:=BB2)

	(*NE - DINT - jämför stack med konstant*)
(*1-1*)
	LD DINT#1
	NE DINT#1
	ST BB2
	CAL PRINT_S(output:="?? false == ")
	CAL PRINTLN_B(output:=BB2)
(*2147483647 - 2147483647*)
	LD DINT#2147483647
	NE DINT#2147483647
	ST BB2
	CAL PRINT_S(output:="?? false == ")
	CAL PRINTLN_B(output:=BB2)
(*-2147483647 - -2147483647*)
	LD DINT#-2147483647
	NE DINT#-2147483647
	ST BB2
	CAL PRINT_S(output:="?? false == ")
	CAL PRINTLN_B(output:=BB2)
(*2147483647 - 0*)
	LD DINT#2147483647
	NE DINT#0
	ST BB2
	CAL PRINT_S(output:="?? true == ")
	CAL PRINTLN_B(output:=BB2)
(*-2147483647 - 0*)
	LD DINT#-2147483647
	NE DINT#0
	ST BB2
	CAL PRINT_S(output:="?? true == ")
	CAL PRINTLN_B(output:=BB2)
(*0 - -2147483647*)
	LD DINT#0
	NE DINT#-2147483647
	ST BB2
	CAL PRINT_S(output:="?? true == ")
	CAL PRINTLN_B(output:=BB2)
(*0 - 2147483647*)
	LD DINT#0
	NE DINT#2147483647
	ST BB2
	CAL PRINT_S(output:="?? true == ")
	CAL PRINTLN_B(output:=BB2)

	(*NE - REAL - jämför stack med variabel*)
	CAL PRINTLN_S(output:="NE - REAL")
(*1.0 - 1.0*)
	LD REAL#1.0
	ST RR1
	LD REAL#1.0
	NE RR1
	ST BB2
	CAL PRINT_S(output:="?? false == ")
	CAL PRINTLN_B(output:=BB2)
(*3.4028235E38 - 3.4028235E38*)
	LD REAL#3.4028235E38
	ST RR1
	LD REAL#3.4028235E38
	NE RR1
	ST BB2
	CAL PRINT_S(output:="?? false == ")
	CAL PRINTLN_B(output:=BB2)
(*1.4E-45 - 1.4E-45*)
	LD REAL#1.4E-45
	ST RR1
	LD REAL#1.4E-45
	NE RR1
	ST BB2
	CAL PRINT_S(output:="?? false == ")
	CAL PRINTLN_B(output:=BB2)
(*0 - 3.4028235E38*)
	LD REAL#3.4028235E38
	ST RR1
	LD REAL#0.0
	NE RR1
	ST BB2
	CAL PRINT_S(output:="?? true == ")
	CAL PRINTLN_B(output:=BB2)
(*0 - 1.4E-45*)
	LD REAL#1.4E-45
	ST RR1
	LD REAL#0.0
	NE RR1
	ST BB2
	CAL PRINT_S(output:="?? true == ")
	CAL PRINTLN_B(output:=BB2)
(*1.4E-45 - 0*)
	LD REAL#0.0
	ST RR1
	LD REAL#1.4E-45
	NE RR1
	ST BB2
	CAL PRINT_S(output:="?? true == ")
	CAL PRINTLN_B(output:=BB2)
(*3.4028235E38 - 0*)
	LD REAL#0.0
	ST RR1
	LD REAL#3.4028235E38
	NE RR1
	ST BB2
	CAL PRINT_S(output:="?? true == ")
	CAL PRINTLN_B(output:=BB2)

	(*NE - REAL - jämför stack med konstant*)
(*1-1*)
	LD REAL#1.0
	NE REAL#1.0
	ST BB2
	CAL PRINT_S(output:="?? false == ")
	CAL PRINTLN_B(output:=BB2)
(*3.4028235E38 - 3.4028235E38*)
	LD REAL#3.4028235E38
	NE REAL#3.4028235E38
	ST BB2
	CAL PRINT_S(output:="?? false == ")
	CAL PRINTLN_B(output:=BB2)
(*1.4E-45 - 1.4E-45*)
	LD REAL#1.4E-45
	NE REAL#1.4E-45
	ST BB2
	CAL PRINT_S(output:="?? false == ")
	CAL PRINTLN_B(output:=BB2)
(*3.4028235E38 - 0*)
	LD REAL#3.4028235E38
	NE REAL#0.0
	ST BB2
	CAL PRINT_S(output:="?? true == ")
	CAL PRINTLN_B(output:=BB2)
(*1.4E-45 - 0*)
	LD REAL#1.4E-45
	NE REAL#0.0
	ST BB2
	CAL PRINT_S(output:="?? true == ")
	CAL PRINTLN_B(output:=BB2)
(*0 - 1.4E-45*)
	LD REAL#0.0
	NE REAL#1.4E-45
	ST BB2
	CAL PRINT_S(output:="?? true == ")
	CAL PRINTLN_B(output:=BB2)
(*0 - 3.4028235E38*)
	LD REAL#0.0
	NE REAL#3.4028235E38
	ST BB2
	CAL PRINT_S(output:="?? true == ")
	CAL PRINTLN_B(output:=BB2)

END_PROGRAM

(* ---- eqtest.il ---- *)
(*
Skall testa EQ
*)
PROGRAM EQtest
   VAR
	BB1, BB2, BB3 : BOOL;
	DD1, DD2, DD3 : DINT;
	RR1, RR2, RR3 : REAL;
	WW1, WW2, WW3 : WSTRING;
   END_VAR
   VAR
	(*Printing*)
	WPrintln : PrintlnWSTRING;
	DPrintln : PrintlnDINT;
	BPrintln : PrintlnBOOL;
	RPrintln : PrintlnREAL;
	WPrint   : PrintWSTRING;
	DPrint   : PrintDINT;
	BPrint   : PrintBOOL;
	RPrint   : PrintREAL;
   END_VAR

	(*BOOL- jämför stack med variabel*)
(*T-T*)
	LD TRUE
	ST BB1
	LD TRUE
	EQ BB1
	ST BB2
	CAL WPrint("?? true == ")
	CAL BPrintln(BB2)

(*T-F*)
	LD FALSE
	ST BB1
	LD TRUE
	EQ BB1
	ST BB2
	CAL WPrint("?? false == ")
	CAL BPrintln(BB2)

(*F-T*)
	LD TRUE
	ST BB1
	LD FALSE
	EQ BB1
	ST BB2
	CAL WPrint("?? false == ")
	CAL BPrintln(BB2)

(*F-F*)
	LD FALSE
	ST BB1
	LD FALSE
	EQ BB1
	ST BB2
	CAL WPrint("?? true == ")
	CAL BPrintln(BB2)

	(*BOOL- jämför stack med konstant*)
(*T-T*)
	LD TRUE
	EQ TRUE
	ST BB2
	CAL WPrint("?? true == ")
	CAL BPrintln(BB2)

(*T-F*)
	LD FALSE
	EQ TRUE
	ST BB2
	CAL WPrint("?? false == ")
	CAL BPrintln(BB2)

(*F-T*)
	LD FALSE
	EQ TRUE
	ST BB2
	CAL WPrint("?? false == ")
	CAL BPrintln(BB2)

(*F-F*)
	LD FALSE
	ST BB1
	LD FALSE
	EQ BB1
	ST BB2
	CAL WPrint("?? true == ")
	CAL BPrintln(BB2)

END_PROGRAM

(*JAVA_BLOCKS for printing (no newline)*)
(*=====================================*)

JAVA_BLOCK JPrintWSTRING
	VAR_IN_OUT
		output: WSTRING;
	END_VAR
END_JAVA_BLOCK
FUNCTION_BLOCK PrintWSTRING
	VAR_IN_OUT
		output: WSTRING;
	END_VAR
	VAR
		jblock: JPrintWSTRING;
	END_VAR
	LD output
	ST jblock.output
	CAL jblock
END_FUNCTION_BLOCK

JAVA_BLOCK JPrintDINT
	VAR_IN_OUT
		output: DINT;
	END_VAR
END_JAVA_BLOCK
FUNCTION_BLOCK PrintDINT
	VAR_IN_OUT
		output: DINT;
	END_VAR
	VAR
		jblock: JPrintDINT;
	END_VAR
	LD output
	ST jblock.output
	CAL jblock
END_FUNCTION_BLOCK
JAVA_BLOCK JPrintREAL
	VAR_IN_OUT
		output:REAL;
	END_VAR
END_JAVA_BLOCK
FUNCTION_BLOCK PrintREAL
	VAR_IN_OUT
		output:REAL;
	END_VAR
	VAR
		jblock:JPrintREAL;
	END_VAR
	LD output
	ST jblock.output
	CAL jblock
END_FUNCTION_BLOCK

JAVA_BLOCK JPrintBOOL
	VAR_IN_OUT
		output: BOOL;
	END_VAR
END_JAVA_BLOCK
FUNCTION_BLOCK PrintBOOL
	VAR_IN_OUT
		output: BOOL;
	END_VAR
	VAR
		jblock: JPrintBOOL;
	END_VAR
	LD output
	ST jblock.output
	CAL jblock
END_FUNCTION_BLOCK

(*JAVA_BLOCKS for printing (newline)*)
(*=====================================*)

JAVA_BLOCK JPrintlnWSTRING
	VAR_IN_OUT
		output: WSTRING;
	END_VAR
END_JAVA_BLOCK
FUNCTION_BLOCK PrintlnWSTRING
	VAR_IN_OUT
		output: WSTRING;
	END_VAR
	VAR
		jblock: JPrintlnWSTRING;
	END_VAR
	LD output
	ST jblock.output
	CAL jblock
END_FUNCTION_BLOCK

JAVA_BLOCK JPrintlnDINT
	VAR_IN_OUT
		output: DINT;
	END_VAR
END_JAVA_BLOCK
FUNCTION_BLOCK PrintlnDINT
	VAR_IN_OUT
		output: DINT;
	END_VAR
	VAR
		jblock: JPrintlnDINT;
	END_VAR
	LD output
	ST jblock.output
	CAL jblock
END_FUNCTION_BLOCK

JAVA_BLOCK JPrintlnREAL
	VAR_IN_OUT
		output:REAL;
	END_VAR
END_JAVA_BLOCK
FUNCTION_BLOCK PrintlnREAL
	VAR_IN_OUT
		output:REAL;
	END_VAR
	VAR
		jblock:JPrintlnREAL;
	END_VAR
	LD output
	ST jblock.output
	CAL jblock
END_FUNCTION_BLOCK

JAVA_BLOCK JPrintlnBOOL
	VAR_IN_OUT
		output: BOOL;
	END_VAR
END_JAVA_BLOCK
FUNCTION_BLOCK PrintlnBOOL
	VAR_IN_OUT
		output: BOOL;
	END_VAR
	VAR
		jblock: JPrintlnBOOL;
	END_VAR
	LD output
	ST jblock.output
	CAL jblock
END_FUNCTION_BLOCK

(* ---- jmptest.il ---- *)
(*This program was run successfully by Anders on thursday 25 April 09:00*)
PROGRAM Jmptest
   VAR
      A : BOOL;
   END_VAR
   VAR
	(*Printing*)
	WPrintln : PrintlnWSTRING;
	DPrintln : PrintlnDINT;
	BPrintln : PrintlnBOOL;
	RPrintln : PrintlnREAL;
	WPrint   : PrintWSTRING;
	DPrint   : PrintDINT;
	BPrint   : PrintBOOL;
	RPrint   : PrintREAL;
   END_VAR

CAL WPrintln("Basic tests....")

(*Test: JMP*)
(*===========*)
    LD TRUE
    JMP e1
        CAL WPrintln("Error")
e1:
    CAL WPrintln("JMP OK")
    (*Check that TRUE remains in resultregister*)
    ST A
	CAL WPrint("OK if true:")
	CAL BPrintln(A)

(*Test: JMPC*)
    (*True should be on the stack*)
    JMPC e2
        CAL WPrintln("Error: JMPC")
e2:
    ST A
	CAL WPrint("OK if true:")
	CAL BPrintln(A)

(*Test: JMPCN*)
    (*True should be on the stack*)
    JMPCN e3
	CAL WPrintln("JMPCN OK")
e3:
(*-------------------------*)
(*Reversed tests*)
(*Expected output:
	JMPC  OK
	JMPCN OK
*)
CAL WPrintln("Reversed tests....")
    LD FALSE
    JMPC e4
	CAL WPrintln("JMPC OK")
e4:
    (*false in RR*)
    JMPCN e5
        CAL WPrintln("ERROR: JMPCN")
	JMP e6
e5: CAL WPrintln("JMPC OK")
e6:

END_PROGRAM

(*JAVA_BLOCKS for printing (no newline)*)
(*=====================================*)

JAVA_BLOCK JPrintWSTRING
	VAR_IN_OUT
		output: WSTRING;
	END_VAR
END_JAVA_BLOCK
FUNCTION_BLOCK PrintWSTRING
	VAR_IN_OUT
		output: WSTRING;
	END_VAR
	VAR
		jblock: JPrintWSTRING;
	END_VAR
	LD output
	ST jblock.output
	CAL jblock
END_FUNCTION_BLOCK

JAVA_BLOCK JPrintDINT
	VAR_IN_OUT
		output: DINT;
	END_VAR
END_JAVA_BLOCK
FUNCTION_BLOCK PrintDINT
	VAR_IN_OUT
		output: DINT;
	END_VAR
	VAR
		jblock: JPrintDINT;
	END_VAR
	LD output
	ST jblock.output
	CAL jblock
END_FUNCTION_BLOCK
JAVA_BLOCK JPrintREAL
	VAR_IN_OUT
		output:REAL;
	END_VAR
END_JAVA_BLOCK
FUNCTION_BLOCK PrintREAL
	VAR_IN_OUT
		output:REAL;
	END_VAR
	VAR
		jblock:JPrintREAL;
	END_VAR
	LD output
	ST jblock.output
	CAL jblock
END_FUNCTION_BLOCK

JAVA_BLOCK JPrintBOOL
	VAR_IN_OUT
		output: BOOL;
	END_VAR
END_JAVA_BLOCK
FUNCTION_BLOCK PrintBOOL
	VAR_IN_OUT
		output: BOOL;
	END_VAR
	VAR
		jblock: JPrintBOOL;
	END_VAR
	LD output
	ST jblock.output
	CAL jblock
END_FUNCTION_BLOCK

(*JAVA_BLOCKS for printing (newline)*)
(*=====================================*)

JAVA_BLOCK JPrintlnWSTRING
	VAR_IN_OUT
		output: WSTRING;
	END_VAR
END_JAVA_BLOCK
FUNCTION_BLOCK PrintlnWSTRING
	VAR_IN_OUT
		output: WSTRING;
	END_VAR
	VAR
		jblock: JPrintlnWSTRING;
	END_VAR
	LD output
	ST jblock.output
	CAL jblock
END_FUNCTION_BLOCK

JAVA_BLOCK JPrintlnDINT
	VAR_IN_OUT
		output: DINT;
	END_VAR
END_JAVA_BLOCK
FUNCTION_BLOCK PrintlnDINT
	VAR_IN_OUT
		output: DINT;
	END_VAR
	VAR
		jblock: JPrintlnDINT;
	END_VAR
	LD output
	ST jblock.output
	CAL jblock
END_FUNCTION_BLOCK

JAVA_BLOCK JPrintlnREAL
	VAR_IN_OUT
		output:REAL;
	END_VAR
END_JAVA_BLOCK
FUNCTION_BLOCK PrintlnREAL
	VAR_IN_OUT
		output:REAL;
	END_VAR
	VAR
		jblock:JPrintlnREAL;
	END_VAR
	LD output
	ST jblock.output
	CAL jblock
END_FUNCTION_BLOCK

JAVA_BLOCK JPrintlnBOOL
	VAR_IN_OUT
		output: BOOL;
	END_VAR
END_JAVA_BLOCK
FUNCTION_BLOCK PrintlnBOOL
	VAR_IN_OUT
		output: BOOL;
	END_VAR
	VAR
		jblock: JPrintlnBOOL;
	END_VAR
	LD output
	ST jblock.output
	CAL jblock
END_FUNCTION_BLOCK

(* ---- logictest.il ---- *)
(*JAVA_BLOCKS for printing (no newline)*)
(*=====================================*)

JAVA_BLOCK JPrintWSTRING
	VAR_IN_OUT
		output: WSTRING;
	END_VAR
END_JAVA_BLOCK
FUNCTION_BLOCK PrintWSTRING
	VAR_IN_OUT
		output: WSTRING;
	END_VAR
	VAR
		jblock: JPrintWSTRING;
	END_VAR
	LD output
	ST jblock.output
	CAL jblock
END_FUNCTION_BLOCK

JAVA_BLOCK JPrintDINT
	VAR_IN_OUT
		output: DINT;
	END_VAR
END_JAVA_BLOCK
FUNCTION_BLOCK PrintDINT
	VAR_IN_OUT
		output: DINT;
	END_VAR
	VAR
		jblock: JPrintDINT;
	END_VAR
	LD output
	ST jblock.output
	CAL jblock
END_FUNCTION_BLOCK
JAVA_BLOCK JPrintREAL
	VAR_IN_OUT
		output:REAL;
	END_VAR
END_JAVA_BLOCK
FUNCTION_BLOCK PrintREAL
	VAR_IN_OUT
		output:REAL;
	END_VAR
	VAR
		jblock:JPrintREAL;
	END_VAR
	LD output
	ST jblock.output
	CAL jblock
END_FUNCTION_BLOCK

JAVA_BLOCK JPrintBOOL
	VAR_IN_OUT
		output: BOOL;
	END_VAR
END_JAVA_BLOCK
FUNCTION_BLOCK PrintBOOL
	VAR_IN_OUT
		output: BOOL;
	END_VAR
	VAR
		jblock: JPrintBOOL;
	END_VAR
	LD output
	ST jblock.output
	CAL jblock
END_FUNCTION_BLOCK

(*JAVA_BLOCKS for printing (newline)*)
(*=====================================*)

JAVA_BLOCK JPrintlnWSTRING
	VAR_IN_OUT
		output: WSTRING;
	END_VAR
END_JAVA_BLOCK
FUNCTION_BLOCK PrintlnWSTRING
	VAR_IN_OUT
		output: WSTRING;
	END_VAR
	VAR
		jblock: JPrintlnWSTRING;
	END_VAR
	LD output
	ST jblock.output
	CAL jblock
END_FUNCTION_BLOCK

JAVA_BLOCK JPrintlnDINT
	VAR_IN_OUT
		output: DINT;
	END_VAR
END_JAVA_BLOCK
FUNCTION_BLOCK PrintlnDINT
	VAR_IN_OUT
		output: DINT;
	END_VAR
	VAR
		jblock: JPrintlnDINT;
	END_VAR
	LD output
	ST jblock.output
	CAL jblock
END_FUNCTION_BLOCK

JAVA_BLOCK JPrintlnREAL
	VAR_IN_OUT
		output:REAL;
	END_VAR
END_JAVA_BLOCK
FUNCTION_BLOCK PrintlnREAL
	VAR_IN_OUT
		output:REAL;
	END_VAR
	VAR
		jblock:JPrintlnREAL;
	END_VAR
	LD output
	ST jblock.output
	CAL jblock
END_FUNCTION_BLOCK

JAVA_BLOCK JPrintlnBOOL
	VAR_IN_OUT
		output: BOOL;
	END_VAR
END_JAVA_BLOCK
FUNCTION_BLOCK PrintlnBOOL
	VAR_IN_OUT
		output: BOOL;
	END_VAR
	VAR
		jblock: JPrintlnBOOL;
	END_VAR
	LD output
	ST jblock.output
	CAL jblock
END_FUNCTION_BLOCK

(*=============================================================*)
(*=============================================================*)
(* Resultat:
	Titta vid XXX kommentarer för att hitta fel
   Innehåll:
     Test1
	Program LOGICtest: test av AND, ANDN, OR
*)

(*Test1*)
PROGRAM LOGICtest
	VAR
		WSpln : PrintlnWSTRING;
		Dpln  : PrintlnDINT;
		Rpln  : PrintlnREAL;
		Bpln  : PrintlnBOOL;
		WSp   : PrintWSTRING;
		Dp    : PrintDINT;
		Rp    : PrintREAL;
		Bp    : PrintBOOL;
	END_VAR
   VAR
	FVAR, TVAR : BOOL;
	RV1, RV2 : BOOL;
	WW1, WW2 : WSTRING;
   END_VAR
(*BOOL*)
(*====*)

LD FALSE
ST FVAR
LD TRUE
ST TVAR

(*pre: FVAR = FALSE, TVAR = FALSE*)
(*AND-operatorn, operand: variabel*)
	CAL WSpln(output:="Test av AND operatorn")
	(*T-T*)
	LD FALSE
	ST RV1
	LD TRUE
	ST RV2 (*end init*)
	LD TRUE

	AND TVAR
	ST  RV1
	ST  RV2

	CAL WSp(output := "?? true == ")
	CAL Bp(output := RV1)
	CAL WSp(output := " ")
	CAL Bpln(output := RV2)

	(*T-F*)
	LD FALSE
	ST RV1
	LD TRUE
	ST RV2 (*end init*)
	LD TRUE

	AND FVAR
	ST  RV1
	ST  RV2

	CAL WSp(output := "?? false == ")
	CAL Bp(output := RV1)
	CAL WSp(output := " ")
	CAL Bpln(output := RV2)

	(*F-T*)
	LD FALSE
	ST RV1
	LD TRUE
	ST RV2 (*end init*)
	LD FALSE

	AND TVAR
	ST  RV1
	ST  RV2

	CAL WSp(output := "?? false == ")
	CAL Bp(output := RV1)
	CAL WSp(output := " ")
	CAL Bpln(output := RV2)

	(*F-F*)
	LD FALSE
	ST RV1
	LD TRUE
	ST RV2 (*end init*)
	LD FALSE

	AND FVAR
	ST  RV1
	ST  RV2

	CAL WSp(output := "?? false == ")
	CAL Bp(output := RV1)
	CAL WSp(output := " ")
	CAL Bpln(output := RV2)

(*pre: FVAR = FALSE, TVAR = FALSE*)
(*AND-operatorn, operand: konstant*)
	CAL WSpln(output:="Test av AND operatorn")
	(*T-T*)
	LD FALSE
	ST RV1
	LD TRUE
	ST RV2 (*end init*)
	LD TRUE

	AND TRUE
	ST  RV1
	ST  RV2

	CAL WSp(output := "?? true == ")
	CAL Bp(output := RV1)
	CAL WSp(output := " ")
	CAL Bpln(output := RV2)

	(*T-F*)
	LD FALSE
	ST RV1
	LD TRUE
	ST RV2 (*end init*)
	LD TRUE

	AND FALSE
	ST  RV1
	ST  RV2

	CAL WSp(output := "?? false == ")
	CAL Bp(output := RV1)
	CAL WSp(output := " ")
	CAL Bpln(output := RV2)

	(*F-T*)
	LD FALSE
	ST RV1
	LD TRUE
	ST RV2 (*end init*)
	LD FALSE

	AND TRUE
	ST  RV1
	ST  RV2

	CAL WSp(output := "?? false == ")
	CAL Bp(output := RV1)
	CAL WSp(output := " ")
	CAL Bpln(output := RV2)

	(*F-F*)
	LD FALSE
	ST RV1
	LD TRUE
	ST RV2 (*end init*)
	LD FALSE

	AND FALSE
	ST  RV1
	ST  RV2

	CAL WSp(output := "?? false == ")
	CAL Bp(output := RV1)
	CAL WSp(output := " ")
	CAL Bpln(output := RV2)

(*pre: FVAR = FALSE, TVAR = FALSE*)
(*OR-operatorn, operand: variabel*)
	CAL WSpln(output:="Test av OR operatorn")
	(*T-T*)
	LD FALSE
	ST RV1
	LD TRUE
	ST RV2 (*end init*)
	LD TRUE

	OR TVAR
	ST  RV1
	ST  RV2

	CAL WSp(output := "?? true == ")
	CAL Bp(output := RV1)
	CAL WSp(output := " ")
	CAL Bpln(output := RV2)

	(*T-F*)
	LD FALSE
	ST RV1
	LD TRUE
	ST RV2 (*end init*)
	LD TRUE

	OR FVAR
	ST  RV1
	ST  RV2

	CAL WSp(output := "?? true == ")
	CAL Bp(output := RV1)
	CAL WSp(output := " ")
	CAL Bpln(output := RV2)

	(*F-T*)
	LD FALSE
	ST RV1
	LD TRUE
	ST RV2 (*end init*)
	LD FALSE

	OR TVAR
	ST  RV1
	ST  RV2

	CAL WSp(output := "?? true == ")
	CAL Bp(output := RV1)
	CAL WSp(output := " ")
	CAL Bpln(output := RV2)

	(*F-F*)
	LD FALSE
	ST RV1
	LD TRUE
	ST RV2 (*end init*)
	LD FALSE

	OR FVAR
	ST  RV1
	ST  RV2

	CAL WSp(output := "?? false == ")
	CAL Bp(output := RV1)
	CAL WSp(output := " ")
	CAL Bpln(output := RV2)

(*pre: FVAR = FALSE, TVAR = FALSE*)
(*OR-operatorn, operand: konstant*)
	CAL WSpln(output:="Test av OR operatorn")
	(*T-T*)
	LD FALSE
	ST RV1
	LD TRUE
	ST RV2 (*end init*)
	LD TRUE

	OR  TRUE
	ST  RV1
	ST  RV2

	CAL WSp(output := "?? true == ")
	CAL Bp(output := RV1)
	CAL WSp(output := " ")
	CAL Bpln(output := RV2)

	(*T-F*)
	LD FALSE
	ST RV1
	LD TRUE
	ST RV2 (*end init*)
	LD TRUE

	OR  FALSE
	ST  RV1
	ST  RV2

	CAL WSp(output := "?? true  == ")
	CAL Bp(output := RV1)
	CAL WSp(output := " ")
	CAL Bpln(output := RV2)

	(*F-T*)
	LD FALSE
	ST RV1
	LD TRUE
	ST RV2 (*end init*)
	LD FALSE

	OR  TRUE
	ST  RV1
	ST  RV2

	CAL WSp(output := "?? true  == ")
	CAL Bp(output := RV1)
	CAL WSp(output := " ")
	CAL Bpln(output := RV2)

	(*F-F*)
	LD FALSE
	ST RV1
	LD TRUE
	ST RV2 (*end init*)
	LD FALSE

	OR  FALSE
	ST  RV1
	ST  RV2

	CAL WSp(output := "?? false == ")
	CAL Bp(output := RV1)
	CAL WSp(output := " ")
	CAL Bpln(output := RV2)

(*pre: FVAR = FALSE, TVAR = FALSE*)
(*ANDN-operatorn, operand: variabel*)
	CAL WSpln(output:="Test av ANDN operatorn")
	(*T-T*)
	LD FALSE
	ST RV1
	LD TRUE
	ST RV2 (*end init*)
	LD TRUE

	ANDN TVAR
	ST  RV1
	ST  RV2

	CAL WSp(output := "?? false == ")
	CAL Bp(output := RV1)
	CAL WSp(output := " ")
	CAL Bpln(output := RV2)

	(*T-F*)
	LD FALSE
	ST RV1
	LD TRUE
	ST RV2 (*end init*)
	LD TRUE

	ANDN FVAR
	ST  RV1
	ST  RV2

	CAL WSp(output := "?? true == ")
	CAL Bp(output := RV1)
	CAL WSp(output := " ")
	CAL Bpln(output := RV2)

	(*F-T*)
	LD FALSE
	ST RV1
	LD TRUE
	ST RV2 (*end init*)
	LD FALSE

	ANDN TVAR
	ST  RV1
	ST  RV2

	CAL WSp(output := "?? false == ")
	CAL Bp(output := RV1)
	CAL WSp(output := " ")
	CAL Bpln(output := RV2)

	(*F-F*)
	LD FALSE
	ST RV1
	LD TRUE
	ST RV2 (*end init*)
	LD FALSE

	ANDN FVAR
	ST  RV1
	ST  RV2

	CAL WSp(output := "?? false == ")
	CAL Bp(output := RV1)
	CAL WSp(output := " ")
	CAL Bpln(output := RV2)

(*pre: FVAR = FALSE, TVAR = FALSE*)
(*ANDN-operatorn, operand: konstant*)
	CAL WSpln(output:="Test av ANDN operatorn")
	(*T-T*)
	LD FALSE
	ST RV1
	LD TRUE
	ST RV2 (*end init*)
	LD TRUE

	ANDN TRUE
	ST  RV1
	ST  RV2

	CAL WSp(output := "?? false == ")
	CAL Bp(output := RV1)
	CAL WSp(output := " ")
	CAL Bpln(output := RV2)

	(*T-F*)
	LD FALSE
	ST RV1
	LD TRUE
	ST RV2 (*end init*)
	LD TRUE

	ANDN FALSE
	ST  RV1
	ST  RV2

	CAL WSp(output := "?? true == ")
	CAL Bp(output := RV1)
	CAL WSp(output := " ")
	CAL Bpln(output := RV2)

	(*F-T*)
	LD FALSE
	ST RV1
	LD TRUE
	ST RV2 (*end init*)
	LD FALSE

	ANDN TRUE
	ST  RV1
	ST  RV2

	CAL WSp(output := "?? false == ")
	CAL Bp(output := RV1)
	CAL WSp(output := " ")
	CAL Bpln(output := RV2)

	(*F-F*)
	LD FALSE
	ST RV1
	LD TRUE
	ST RV2 (*end init*)
	LD FALSE

	ANDN FALSE
	ST  RV1
	ST  RV2

	CAL WSp(output := "?? false == ")
	CAL Bp(output := RV1)
	CAL WSp(output := " ")
	CAL Bpln(output := RV2)

(*pre: FVAR = FALSE, TVAR = FALSE*)
(*ORN-operatorn, operand: variabel*)
	CAL WSpln(output:="Test av ORN operatorn")
	(*T-T*)
	LD FALSE
	ST RV1
	LD TRUE
	ST RV2 (*end init*)
	LD TRUE

	ORN TVAR
	ST  RV1
	ST  RV2

	CAL WSp(output := "?? true  == ")
	CAL Bp(output := RV1)
	CAL WSp(output := " ")
	CAL Bpln(output := RV2)

	(*T-F*)
	LD FALSE
	ST RV1
	LD TRUE
	ST RV2 (*end init*)
	LD TRUE

	ORN FVAR
	ST  RV1
	ST  RV2

	CAL WSp(output := "?? true  == ")
	CAL Bp(output := RV1)
	CAL WSp(output := " ")
	CAL Bpln(output := RV2)

	(*F-T*)
	LD FALSE
	ST RV1
	LD TRUE
	ST RV2 (*end init*)
	LD FALSE

	ORN TVAR
	ST  RV1
	ST  RV2

	CAL WSp(output := "?? false == ")
	CAL Bp(output := RV1)
	CAL WSp(output := " ")
	CAL Bpln(output := RV2)

	(*F-F*)
	LD FALSE
	ST RV1
	LD TRUE
	ST RV2 (*end init*)
	LD FALSE

	ORN FVAR
	ST  RV1
	ST  RV2

	CAL WSp(output := "?? true  == ")
	CAL Bp(output := RV1)
	CAL WSp(output := " ")
	CAL Bpln(output := RV2)

(*pre: FVAR = FALSE, TVAR = FALSE*)
(*ORN-operatorn, operand: konstant*)
	CAL WSpln(output:="Test av ORN operatorn")
	(*T-T*)
	LD FALSE
	ST RV1
	LD TRUE
	ST RV2 (*end init*)
	LD TRUE

	ORN TRUE
	ST  RV1
	ST  RV2

	CAL WSp(output := "?? true  == ")
	CAL Bp(output := RV1)
	CAL WSp(output := " ")
	CAL Bpln(output := RV2)

	(*T-F*)
	LD FALSE
	ST RV1
	LD TRUE
	ST RV2 (*end init*)
	LD TRUE

	ORN FALSE
	ST  RV1
	ST  RV2

	CAL WSp(output := "?? true  == ")
	CAL Bp(output := RV1)
	CAL WSp(output := " ")
	CAL Bpln(output := RV2)

	(*F-T*)
	LD FALSE
	ST RV1
	LD TRUE
	ST RV2 (*end init*)
	LD FALSE

	ORN TRUE
	ST  RV1
	ST  RV2

	CAL WSp(output := "?? false == ")
	CAL Bp(output := RV1)
	CAL WSp(output := " ")
	CAL Bpln(output := RV2)

	(*F-F*)
	LD FALSE
	ST RV1
	LD TRUE
	ST RV2 (*end init*)
	LD FALSE

	ORN FALSE
	ST  RV1
	ST  RV2

	CAL WSp(output := "?? true  == ")
	CAL Bp(output := RV1)
	CAL WSp(output := " ")
	CAL Bpln(output := RV2)

(*pre: FVAR = FALSE, TVAR = FALSE*)
(*XOR-operatorn, operand: variabel*)
	CAL WSpln(output:="Test av XOR operatorn")
	(*T-T*)
	LD FALSE
	ST RV1
	LD TRUE
	ST RV2 (*end init*)
	LD TRUE

	XOR TVAR
	ST  RV1
	ST  RV2

	CAL WSp(output := "?? false == ")
	CAL Bp(output := RV1)
	CAL WSp(output := " ")
	CAL Bpln(output := RV2)

	(*T-F*)
	LD FALSE
	ST RV1
	LD TRUE
	ST RV2 (*end init*)
	LD TRUE

	XOR FVAR
	ST  RV1
	ST  RV2

	CAL WSp(output := "?? true  == ")
	CAL Bp(output := RV1)
	CAL WSp(output := " ")
	CAL Bpln(output := RV2)

	(*F-T*)
	LD FALSE
	ST RV1
	LD TRUE
	ST RV2 (*end init*)
	LD FALSE

	XOR TVAR
	ST  RV1
	ST  RV2

	CAL WSp(output := "?? true  == ")
	CAL Bp(output := RV1)
	CAL WSp(output := " ")
	CAL Bpln(output := RV2)

	(*F-F*)
	LD FALSE
	ST RV1
	LD TRUE
	ST RV2 (*end init*)
	LD FALSE

	XOR FVAR
	ST  RV1
	ST  RV2

	CAL WSp(output := "?? false == ")
	CAL Bp(output := RV1)
	CAL WSp(output := " ")
	CAL Bpln(output := RV2)

(*pre: FVAR = FALSE, TVAR = FALSE*)
(*XOR-operatorn, operand: konstant*)
	CAL WSpln(output:="Test av XOR operatorn")
	(*T-T*)
	LD FALSE
	ST RV1
	LD TRUE
	ST RV2 (*end init*)
	LD TRUE

	XOR TRUE
	ST  RV1
	ST  RV2

	CAL WSp(output := "?? false == ")
	CAL Bp(output := RV1)
	CAL WSp(output := " ")
	CAL Bpln(output := RV2)

	(*T-F*)
	LD FALSE
	ST RV1
	LD TRUE
	ST RV2 (*end init*)
	LD TRUE

	XOR FALSE
	ST  RV1
	ST  RV2

	CAL WSp(output := "?? true  == ")
	CAL Bp(output := RV1)
	CAL WSp(output := " ")
	CAL Bpln(output := RV2)

	(*F-T*)
	LD FALSE
	ST RV1
	LD TRUE
	ST RV2 (*end init*)
	LD FALSE

	XOR TRUE
	ST  RV1
	ST  RV2

	CAL WSp(output := "?? true  == ")
	CAL Bp(output := RV1)
	CAL WSp(output := " ")
	CAL Bpln(output := RV2)

	(*F-F*)
	LD FALSE
	ST RV1
	LD TRUE
	ST RV2 (*end init*)
	LD FALSE

	XOR FALSE
	ST  RV1
	ST  RV2

	CAL WSp(output := "?? false == ")
	CAL Bp(output := RV1)
	CAL WSp(output := " ")
	CAL Bpln(output := RV2)

(*pre: FVAR = FALSE, TVAR = FALSE*)
(*XORN-operatorn, operand: variabel*)
	CAL WSpln(output:="Test av XORN operatorn")
	(*T-T*)
	LD FALSE
	ST RV1
	LD TRUE
	ST RV2 (*end init*)
	LD TRUE

	XORN TVAR
	ST  RV1
	ST  RV2

	CAL WSp(output := "?? true  == ")
	CAL Bp(output := RV1)
	CAL WSp(output := " ")
	CAL Bpln(output := RV2)

	(*T-F*)
	LD FALSE
	ST RV1
	LD TRUE
	ST RV2 (*end init*)
	LD TRUE

	XORN FVAR
	ST  RV1
	ST  RV2

	CAL WSp(output := "?? false == ")
	CAL Bp(output := RV1)
	CAL WSp(output := " ")
	CAL Bpln(output := RV2)

	(*F-T*)
	LD FALSE
	ST RV1
	LD TRUE
	ST RV2 (*end init*)
	LD FALSE

	XORN TVAR
	ST  RV1
	ST  RV2

	CAL WSp(output := "?? false == ")
	CAL Bp(output := RV1)
	CAL WSp(output := " ")
	CAL Bpln(output := RV2)

	(*F-F*)
	LD FALSE
	ST RV1
	LD TRUE
	ST RV2 (*end init*)
	LD FALSE

	XORN FVAR
	ST  RV1
	ST  RV2

	CAL WSp(output := "?? true  == ")
	CAL Bp(output := RV1)
	CAL WSp(output := " ")
	CAL Bpln(output := RV2)

(*pre: FVAR = FALSE, TVAR = FALSE*)
(*XORN-operatorn, operand: konstant*)
	CAL WSpln(output:="Test av XORN operatorn")
	(*T-T*)
	LD FALSE
	ST RV1
	LD TRUE
	ST RV2 (*end init*)
	LD TRUE

	XORN TRUE
	ST  RV1
	ST  RV2

	CAL WSp(output := "?? true  == ")
	CAL Bp(output := RV1)
	CAL WSp(output := " ")
	CAL Bpln(output := RV2)

	(*T-F*)
	LD FALSE
	ST RV1
	LD TRUE
	ST RV2 (*end init*)
	LD TRUE

	XORN FALSE
	ST  RV1
	ST  RV2

	CAL WSp(output := "?? false == ")
	CAL Bp(output := RV1)
	CAL WSp(output := " ")
	CAL Bpln(output := RV2)

	(*F-T*)
	LD FALSE
	ST RV1
	LD TRUE
	ST RV2 (*end init*)
	LD FALSE

	XORN TRUE
	ST  RV1
	ST  RV2

	CAL WSp(output := "?? false == ")
	CAL Bp(output := RV1)
	CAL WSp(output := " ")
	CAL Bpln(output := RV2)

	(*F-F*)
	LD FALSE
	ST RV1
	LD TRUE
	ST RV2 (*end init*)
	LD FALSE

	XORN FALSE
	ST  RV1
	ST  RV2

	CAL WSp(output := "?? true  == ")
	CAL Bp(output := RV1)
	CAL WSp(output := " ")
	CAL Bpln(output := RV2)

END_PROGRAM

(* ---- variablefbtest.il ---- *)
(*JAVA_BLOCKS for printing (no newline)*)
(*=====================================*)

JAVA_BLOCK JPrintWSTRING
	VAR_IN_OUT
		output: WSTRING;
	END_VAR
END_JAVA_BLOCK
FUNCTION_BLOCK PrintWSTRING
	VAR_IN_OUT
		output: WSTRING;
	END_VAR
	VAR
		jblock: JPrintWSTRING;
	END_VAR
	LD output
	ST jblock.output
	CAL jblock
END_FUNCTION_BLOCK

JAVA_BLOCK JPrintDINT
	VAR_IN_OUT
		output: DINT;
	END_VAR
END_JAVA_BLOCK
FUNCTION_BLOCK PrintDINT
	VAR_IN_OUT
		output: DINT;
	END_VAR
	VAR
		jblock: JPrintDINT;
	END_VAR
	LD output
	ST jblock.output
	CAL jblock
END_FUNCTION_BLOCK
JAVA_BLOCK JPrintREAL
	VAR_IN_OUT
		output:REAL;
	END_VAR
END_JAVA_BLOCK
FUNCTION_BLOCK PrintREAL
	VAR_IN_OUT
		output:REAL;
	END_VAR
	VAR
		jblock:JPrintREAL;
	END_VAR
	LD output
	ST jblock.output
	CAL jblock
END_FUNCTION_BLOCK

JAVA_BLOCK JPrintBOOL
	VAR_IN_OUT
		output: BOOL;
	END_VAR
END_JAVA_BLOCK
FUNCTION_BLOCK PrintBOOL
	VAR_IN_OUT
		output: BOOL;
	END_VAR
	VAR
		jblock: JPrintBOOL;
	END_VAR
	LD output
	ST jblock.output
	CAL jblock
END_FUNCTION_BLOCK

(*JAVA_BLOCKS for printing (newline)*)
(*=====================================*)

JAVA_BLOCK JPrintlnWSTRING
	VAR_IN_OUT
		output: WSTRING;
	END_VAR
END_JAVA_BLOCK
FUNCTION_BLOCK PrintlnWSTRING
	VAR_IN_OUT
		output: WSTRING;
	END_VAR
	VAR
		jblock: JPrintlnWSTRING;
	END_VAR
	LD output
	ST jblock.output
	CAL jblock
END_FUNCTION_BLOCK

JAVA_BLOCK JPrintlnDINT
	VAR_IN_OUT
		output: DINT;
	END_VAR
END_JAVA_BLOCK
FUNCTION_BLOCK PrintlnDINT
	VAR_IN_OUT
		output: DINT;
	END_VAR
	VAR
		jblock: JPrintlnDINT;
	END_VAR
	LD output
	ST jblock.output
	CAL jblock
END_FUNCTION_BLOCK

JAVA_BLOCK JPrintlnREAL
	VAR_IN_OUT
		output:REAL;
	END_VAR
END_JAVA_BLOCK
FUNCTION_BLOCK PrintlnREAL
	VAR_IN_OUT
		output:REAL;
	END_VAR
	VAR
		jblock:JPrintlnREAL;
	END_VAR
	LD output
	ST jblock.output
	CAL jblock
END_FUNCTION_BLOCK

JAVA_BLOCK JPrintlnBOOL
	VAR_IN_OUT
		output: BOOL;
	END_VAR
END_JAVA_BLOCK
FUNCTION_BLOCK PrintlnBOOL
	VAR_IN_OUT
		output: BOOL;
	END_VAR
	VAR
		jblock: JPrintlnBOOL;
	END_VAR
	LD output
	ST jblock.output
	CAL jblock
END_FUNCTION_BLOCK

(*=============================================================*)
(*=============================================================*)

FUNCTION_BLOCK LDSTfbfoo
	LD TRUE
END_FUNCTION_BLOCK

FUNCTION_BLOCK LDSTfbtestfb
(*This FB is only a holder of vars, its run method doesn't
  do anything essential*)
   VAR_IN_OUT
	BB1, BB2 : BOOL;
	DD1, DD2 : DINT;
	RR1, RR2 : REAL;
	WW1, WW2 : WSTRING;
	FF : LDSTfbfoo;
   END_VAR
	LD BB1
	ST BB2
	LD DD1
	ST DD2
	LD RR1
	ST RR2
	LD WW1
	ST WW2
END_FUNCTION_BLOCK

PROGRAM LDSTfbtest
	VAR
		WPrintln : PrintlnWSTRING;
		DPrintln  : PrintlnDINT;
		RPrintln  : PrintlnREAL;
		BPrintln  : PrintlnBOOL;
		WPrint   : PrintWSTRING;
		DPrint    : PrintDINT;
		RPrint    : PrintREAL;
		BPrint    : PrintBOOL;
	END_VAR
   VAR
	BB1, BB2 : BOOL;
	DD1, DD2 : DINT;
	RR1, RR2 : REAL;
	WW1, WW2 : WSTRING;
	FB1 : LDSTfbtestfb;
	FB2 : LDSTfbfoo;
   END_VAR

CAL WPrintln("Testing LD & ST of BOOL,DINT,REAL,WSTRING to/from FBs")
   LD TRUE
   ST BB1
   ST FB1.BB1

   LD DINT#1234567890
   ST DD1
   ST FB1.DD1

   LD REAL#123.345
   ST RR1
   ST FB1.RR1

   LD "abcdef"
   ST WW1
   ST FB1.WW1

   CAL FB1

   LD FB1.BB2
   ST BB2
   LD FB1.DD2
   ST DD2
   LD FB1.RR2
   ST RR2
   LD FB1.WW2
   ST WW2

   	CAL WPrint("?? ")
	CAL BPrint(BB1)
	CAL WPrint(" == ")
	CAL BPrintln(BB2)

   	CAL WPrint("?? ")
	CAL DPrint(DD1)
	CAL WPrint(" == ")
	CAL DPrintln(DD2)

   	CAL WPrint("?? ")
	CAL RPrint(RR1)
	CAL WPrint(" == ")
	CAL RPrintln(RR2)

  	CAL WPrint("?? ")
	CAL WPrint(WW1)
	CAL WPrint(" == ")
	CAL WPrintln(WW2)

(* Thomas titta på detta*)

	LD FB2
   	ST FB1.FF
   	LD FB1.FF
   	ST FB2

END_PROGRAM

(* ---- variabletest.il ---- *)
(*JAVA_BLOCKS for printing (no newline)*)
(*=====================================*)

JAVA_BLOCK JPrintWSTRING
	VAR_IN_OUT
		output: WSTRING;
	END_VAR
END_JAVA_BLOCK
FUNCTION_BLOCK PrintWSTRING
	VAR_IN_OUT
		output: WSTRING;
	END_VAR
	VAR
		jblock: JPrintWSTRING;
	END_VAR
	LD output
	ST jblock.output
	CAL jblock
END_FUNCTION_BLOCK

JAVA_BLOCK JPrintDINT
	VAR_IN_OUT
		output: DINT;
	END_VAR
END_JAVA_BLOCK
FUNCTION_BLOCK PrintDINT
	VAR_IN_OUT
		output: DINT;
	END_VAR
	VAR
		jblock: JPrintDINT;
	END_VAR
	LD output
	ST jblock.output
	CAL jblock
END_FUNCTION_BLOCK
JAVA_BLOCK JPrintREAL
	VAR_IN_OUT
		output:REAL;
	END_VAR
END_JAVA_BLOCK
FUNCTION_BLOCK PrintREAL
	VAR_IN_OUT
		output:REAL;
	END_VAR
	VAR
		jblock:JPrintREAL;
	END_VAR
	LD output
	ST jblock.output
	CAL jblock
END_FUNCTION_BLOCK

JAVA_BLOCK JPrintBOOL
	VAR_IN_OUT
		output: BOOL;
	END_VAR
END_JAVA_BLOCK
FUNCTION_BLOCK PrintBOOL
	VAR_IN_OUT
		output: BOOL;
	END_VAR
	VAR
		jblock: JPrintBOOL;
	END_VAR
	LD output
	ST jblock.output
	CAL jblock
END_FUNCTION_BLOCK

(*JAVA_BLOCKS for printing (newline)*)
(*=====================================*)

JAVA_BLOCK JPrintlnWSTRING
	VAR_IN_OUT
		output: WSTRING;
	END_VAR
END_JAVA_BLOCK
FUNCTION_BLOCK PrintlnWSTRING
	VAR_IN_OUT
		output: WSTRING;
	END_VAR
	VAR
		jblock: JPrintlnWSTRING;
	END_VAR
	LD output
	ST jblock.output
	CAL jblock
END_FUNCTION_BLOCK

JAVA_BLOCK JPrintlnDINT
	VAR_IN_OUT
		output: DINT;
	END_VAR
END_JAVA_BLOCK
FUNCTION_BLOCK PrintlnDINT
	VAR_IN_OUT
		output: DINT;
	END_VAR
	VAR
		jblock: JPrintlnDINT;
	END_VAR
	LD output
	ST jblock.output
	CAL jblock
END_FUNCTION_BLOCK

JAVA_BLOCK JPrintlnREAL
	VAR_IN_OUT
		output:REAL;
	END_VAR
END_JAVA_BLOCK
FUNCTION_BLOCK PrintlnREAL
	VAR_IN_OUT
		output:REAL;
	END_VAR
	VAR
		jblock:JPrintlnREAL;
	END_VAR
	LD output
	ST jblock.output
	CAL jblock
END_FUNCTION_BLOCK

JAVA_BLOCK JPrintlnBOOL
	VAR_IN_OUT
		output: BOOL;
	END_VAR
END_JAVA_BLOCK
FUNCTION_BLOCK PrintlnBOOL
	VAR_IN_OUT
		output: BOOL;
	END_VAR
	VAR
		jblock: JPrintlnBOOL;
	END_VAR
	LD output
	ST jblock.output
	CAL jblock
END_FUNCTION_BLOCK

(*=============================================================*)
(*=============================================================*)
(* Resultat:
	Titta vid XXX kommentarer för att hitta fel
   Innehåll:
     Test1
	Program LDSTtest: för att test LD och ST för 4 datatyper

*)

(*Test1*)
PROGRAM LDSTtest
	VAR
		WPrintln : PrintlnWSTRING;
		DPrintln  : PrintlnDINT;
		RPrintln  : PrintlnREAL;
		BPrintln  : PrintlnBOOL;
		WPrint   : PrintWSTRING;
		DPrint    : PrintDINT;
		RPrint    : PrintREAL;
		BPrint    : PrintBOOL;
	END_VAR
   VAR
	BB1, BB2 : BOOL;
	DD1, DD2 : DINT;
	RR1, RR2 : REAL;
	WW1, WW2 : WSTRING;
   END_VAR
(*BOOL*)
(*====*)
   CAL WPrintln("Tests of BOOL constants and variables")
   (*BOOL*)
   LD TRUE
   ST BB1
   CAL WPrint("?? true == ")
   CAL BPrintln(BB1)

   (*BOOL*)
   LD FALSE
   ST BB1
   CAL WPrint("?? false == ")
   CAL BPrintln(BB1)

   (*BOOL*)
   LD BOOL#1
   ST BB1
   CAL WPrint("?? true == ")
   CAL BPrint(BB1)

   (*BOOL*)
   LD BOOL#0
   ST BB1
   CAL WPrint("?? false == ")
   CAL BPrint(BB1)

   (*BOOL*)
   LD TRUE
   ST BB1
   LD BB1
   ST BB2
   CAL WPrint("?? true == ")
   CAL BPrintln(BB2)

   (*BOOL*)
   LD FALSE
   ST BB1
   LD BB1
   ST BB2
   CAL WPrint("?? false == ")
   CAL BPrintln(BB2)

CAL WPrintln("Testing LDN/STN")
   (*LDN/STN finns bara på BOOL*)
   LDN TRUE
   ST  BB1
   CAL WPrint("?? false == ")
   CAL BPrintln(BB1)

   LDN FALSE
   ST  BB1
   CAL WPrint("?? true == ")
   CAL BPrintln(BB1)

   LD  TRUE
   STN BB1
   CAL WPrint("?? false == ")
   CAL BPrintln(BB1)

   LD  TRUE
   STN  BB1
   CAL WPrint("?? false == ")
   CAL BPrintln(BB1)

   LD TRUE
   ST  BB2
   LDN BB2
   ST  BB1
   CAL WPrint("?? false == ")
   CAL BPrintln(BB1)

   LD FALSE
   ST  BB2
   LDN BB2
   ST  BB1
   CAL WPrint("?? true == ")
   CAL BPrintln(BB1)

   LD  TRUE
   STN BB1
   CAL WPrint("?? false == ")
   CAL BPrintln(BB1)

   LD  FALSE
   STN  BB1
   CAL WPrint("?? true == ")
   CAL BPrintln(BB1)

(*Fall som alltid skall ge fel*)
(*
	ST DINT#3
	STN TRUE
*)

(*DINT*)
(*====*)
CAL WPrintln("Tests of DINT constants and variables")
   (*DINT*)
   LD DINT#0
   ST DD1
   CAL WPrint("?? 0 == ")
   CAL DPrintln(DD1)

   (*DINT*)
   LD DINT#-1
   ST DD1
   CAL WPrint("?? -1 == ")
   CAL DPrintln(DD1)

   (*DINT*)
   LD DINT#1
   ST DD1
   CAL WPrint("?? 1 == ")
   CAL DPrintln(DD1)

   (*DINT*)
   LD DINT#23_344
   ST DD1
   CAL WPrint("?? 23344 == ")
   CAL DPrintln(DD1)

   (*DINT: test of binary constants*)
   LD DINT#2#1111_1111
   ST DD1
   CAL WPrint("?? 255 == ")
   CAL DPrintln(DD1)

   LD DINT#2#0000_1000
   ST DD1
   CAL WPrint("?? 8 == ")
   CAL DPrintln(DD1)

   LD DINT#2#0
   ST DD1
   CAL WPrint("?? 0 == ")
   CAL DPrintln(DD1)

   LD DINT#2#11
   ST DD1
   CAL WPrint("?? 3 == ")
   CAL DPrintln(DD1)

   (*DINT: test of octal constants*)
   LD DINT#8#377
   ST DD1
   CAL WPrint("?? 255 == ")
   CAL DPrintln(DD1)

   LD DINT#8#020
   ST DD1
   CAL WPrint("?? 16 == ")
   CAL DPrintln(DD1)

   LD DINT#8#0
   ST DD1
   CAL WPrint("?? 0 == ")
   CAL DPrintln(DD1)

   (*DINT: test of hexadecimal constants*)
   LD DINT#16#FF
   ST DD1
   CAL WPrint("?? 255 == ")
   CAL DPrintln(DD1)

   LD DINT#16#A0
   ST DD1
   CAL WPrint("?? 160 == ")
   CAL DPrintln(DD1)

   LD DINT#16#0
   ST DD1
   CAL WPrint("?? 0 == ")
   CAL DPrintln(DD1)

   (*DINT: test of variables*)
   LD DINT#34
   ST DD1
   LD DD1
   ST DD2
   CAL WPrint("?? 34 == ")
   CAL DPrintln(DD2)

(*REAL*)
(*====*)
CAL WPrintln("Tests of REAL constants and variables")

   LD REAL#0.0
   ST RR1
   CAL WPrint("?? 0 == ")
   CAL RPrintln(RR1)

   LD REAL#12.12
   ST RR1
   CAL WPrint("?? 12.12 == ")
   CAL RPrintln(RR1)

   LD REAL#-12.12
   ST RR1
   CAL WPrint("?? -12.12 == ")
   CAL RPrintln(RR1)

   LD REAL#0.1
   ST RR1
   CAL WPrint("?? 0.1 == ")
   CAL RPrintln(RR1)

   LD REAL#10.123
   ST RR1
   CAL WPrint("?? 10.123 == ")
   CAL RPrintln(RR1)

   LD REAL#+12_123.21
   ST RR1
   CAL WPrint("?? 12123.21 == ")
   CAL RPrintln(RR1)

   LD REAL#-0.001298
   ST RR1
   CAL WPrint("?? -0.001298 == ")
   CAL RPrintln(RR1)

   LD REAL#-1.65E-10
   ST RR1
   CAL WPrint("?? -1.65E-10 == ")
   CAL RPrintln(RR1)

   LD REAL#0.9E20
   ST RR1
   CAL WPrint("?? 0.9E20 == ")
   CAL RPrintln(RR1)

   LD REAL#0.3276e+14
   ST RR1
   CAL WPrint("?? 0.3276e+14== ")
   CAL RPrintln(RR1)

   LD REAL#0.3276e+14
   ST RR1
   LD RR1
   ST RR2
   CAL WPrint("?? 0.3276e+14== ")
   CAL RPrintln(RR2)

(*WSTRING*)
(*=======*)
CAL WPrintln("Tests of WSTRING constants and variables")

   LD "Testing double_byte_character_string"
   ST WW1
   CAL WPrint("?? Testing double_byte_character_string == ")
   CAL WPrintln(WW1)

   LD "åäöÅÄÖ!@#$%^&*()_+|~1" (*234567890-=\`¤{}[]:;$"'<>,.?/"*)
   ST WW1
   CAL WPrintln("?? åäöÅÄÖ!@#$%^&*()_+|~1 == ")
   CAL WPrint("   ")
   CAL WPrintln(WW1)

(*XXX error, see further comments*)
   LD "234567890-=`{}[]:;$"'<>$\,.?/$"
			(* XXX ¤ does not work*)
			(* XXX $\ should print as \
			   XXX $" should print as "
			*)
   ST WW1
   CAL WPrintln("?? 234567890-=`{}[]:;$"'<>$\,.?/$ == ")
   CAL WPrint("   ")
   CAL WPrintln(WW1)

   LD "abcdefghijklmnopqrstuvxyzåäöABCDEFGHIJKLMNOPQRSTUVXYZÅÄÖ"
   ST WW1
   LD WW1
   ST WW2
   CAL WPrintln("?? abcdefghijklmnopqrstuvxyzåäöABCDEFGHIJKLMNOPQRSTUVXYZÅÄÖ == ")
   CAL WPrint("   ")
   CAL WPrintln(WW2)

END_PROGRAM
